(* CODESYS project XPlanarApplication.library
   Company: Beckhoff Automation LLC
   DefaultNamespace: XPlanarApplication
   Version: 1.0.1
   Placeholder: XPlanarApplication
   Title: XPlanarApplication

Project tree, tasks and I/O mapping:
  libraries: SPT Base Types, * (Beckhoff Automation LLC); SPT Event Logger, * (Beckhoff Automation LLC); Tc2_Math, * (Beckhoff Automation GmbH); Tc2_Standard, * (Beckhoff Automation GmbH); Tc2_System, * (Beckhoff Automation GmbH); Tc2_Utilities, * (Beckhoff Automation GmbH); Tc3_EventLogger, * (Beckhoff Automation GmbH); Tc3_Mc3PlanarMotion, * (Beckhoff Automation GmbH); Tc3_Physics, * (Beckhoff Automation GmbH); Tc3_XPlanarUtility, * (Beckhoff Automation GmbH)
  Mover/
    DUTs/
      data type ST_CommandLog
      data type ST_MoveDynamics
      data type ST_MoverCommand
      data type ST_MoverHMI
      data type ST_MoverObjectInfos
    TaskClasses/
      function block FB_AddToGroup [ST]: Execute
      function block FB_Disable [ST]: Execute
      function block FB_Enable [ST]: Execute
      function block FB_Halt [ST]: Execute
      function block FB_JoinClosestTrack [ST]: Execute, Update
      function block FB_JoinTrack [ST]: Execute
      function block FB_LeaveTrack [ST]: Execute
      function block FB_MoveA [ST]: Execute
      function block FB_MoveB [ST]: Execute
      function block FB_MoveToPosition [ST]: Execute
      function block FB_MoveZ [ST]: Execute
      function block FB_ResetMover [ST]: Execute
      function block FB_Rotate [ST]: Execute
      function block FB_SquareUp [ST]: Execute, Update
      function block FB_TrackMove [ST]: Execute
      function block FB_TrackMoveXY [ST]: Execute
    function block FB_XPlanarMover [ST]: FreeMove, JoinClosestTrack, JoinTrack, LeaveTrack, Rotate, SendToStation, SquareUp, TiltA, TiltB, TrackMove, TrackMoveXY, VerticalMove, Movement, Rotation, Tilt, ActualPosition, AddToGroup, CommandLog, Destination, Disable, Dynamics, Enable, Gap, Halt, IdentifiedBTN, InStation, MoveCommand, MoverBTN, MoverIndex, MoverType, pm, Reset, Status, Utility, CyclicLogic
    interface I_MoveCommands: FreeMove, JoinClosestTrack, JoinTrack, LeaveTrack, Rotate, SendToStation, SquareUp, TiltA, TiltB, TrackMove, TrackMoveXY, VerticalMove
    interface I_MoveDynamics: Movement, Rotation, Tilt
    interface I_XPlanarMover: ActualPosition, AddToGroup, CommandLog, Destination, Disable, Dynamics, Enable, Gap, Halt, IdentifiedBTN, InStation, MoveCommand, MoverBTN, MoverIndex, MoverType, pm, Reset, Status, Utility
  Part/
    Tasks/
      function block FB_AllowEnable [ST]: Execute
      function block FB_ForceDisable [ST]: Execute
      function block FB_Initialize [ST]: Execute
      function block FB_ResetPart [ST]: Execute
    function block FB_XPlanarPart [ST]: CyclicLogic, ForceDisable, Initialize, ObjectID, pm, Reset, SetAllowEnable, State
    interface I_XPlanarPart: ForceDisable, ObjectID, pm, Reset, SetAllowEnable, State
  Project Information/
    function F_GetCompany [ST]
    function F_GetTitle [ST]
    function F_GetVersion [ST]
  Station/
    DUT/
      data type E_StationType
      data type E_XplanarStationState
      data type ST_StationHMI
      data type ST_XPlanarStationObjectInfos
    function block FB_MoverQueue [ST]: Clear, Count, Dequeue, Enqueue, FirstMover, LastMover, MoverIDs, Queue
    function block FB_XPlanarStationBase [ST]: AllowQueing, CanReleaseMover, CurrentMover, Error, Execute, HasMover, ID, MoverDetected, MoverQueue, NextStation, NumMoversRequired, Position, Reset, Size, StationComplete, StationReady, StationType, TrackID, CyclicLogic, Name, WatchForMover
    interface I_XPlanarStation: AllowQueing, CanReleaseMover, CurrentMover, Execute, HasMover, ID, MoverQueue, Name, NextStation, NumMoversRequired, Position, Reset, Size, StationComplete, StationReady, StationType, TrackID
  Tile/
    DUT/
      data type ST_TileObjectInfos
      data type ST_TileTemperatures
    function block FB_XPlanarTile [ST]: Btn, CyclicLogic, DcLinkOk, Index, Initialize, PartIndex, PositionOnPart, Temperatures, TimeToShutdown, Update, Utility
    interface I_XPlanarTile: Btn, DcLinkOk, Index, PartIndex, PositionOnPart, Temperatures, TimeToShutdown, Update, Utility
  Track/
    DUT/
      data type E_TrackItemType
      data type ST_TrackDefinition
      data type ST_TrackItems
      data type ST_TrackStatus
    TaskClasses/
      function block FB_AddTrackToGroup [ST]: Execute
      function block FB_AppendLine [ST]: Execute
      function block FB_AppendPoint [ST]: Execute
      function block FB_BuildTrack [ST]: Execute, Update
      function block FB_ClearSegment [ST]: Execute
      function block FB_CloseLoop [ST]: Execute
      function block FB_DisableTrack [ST]: Execute
      function block FB_EnableTrack [ST]: Execute
      function block FB_SetEndAtTrack [ST]: Execute
      function block FB_SetStartFromTrack [ST]: Execute
      function block FB_TrackReset [ST]: Execute
    function block FB_XPlanarTrackSegment [ST]: AddToGroup, AppendLine, AppendPoint, Build, Clear, CloseLoop, Definition, Disable, Enable, GetTrackPositionAt, Index, MoverCount, MovingMoverCount, pm, Reset, SetEndAtTrack, SetStartFromTrack, Status, TrackLength, Utility, CyclicLogic
    interface I_XPlanarTrack: AddToGroup, AppendLine, AppendPoint, Build, Clear, CloseLoop, Definition, Disable, Enable, GetTrackPositionAt, Index, MoverCount, MovingMoverCount, pm, Reset, Status, TrackLength, Utility
  Version/
    global variables Global_Version
  XPlanarComponent/
    TaskClasses/
      function block FB_EnableGroup [ST]: Execute
      function block FB_MoverIdentification [ST]: Execute, Update
      function block FB_MoverRedetection [ST]: Execute, Update
      function block FB_ResetGroup [ST]: Execute
      function block FB_ResetXPlanar [ST]: Execute, Update
    function block FB_Component_XPlanar [ST]: CreateEvents, Monitoring, CyclicLogic, Abort, AddMoversToGroup, AddTracksToGroup, EnableGroup, EnableMovers, EnableTracks, IdentifyMovers, Initialize, MoverDetectionInfo, MoverRedetect, Reset, TileCount, TracksInitialized, Utility
  XPlanarResultClasses/
    function block FB_MoverTaskResult [ST]: Mover, Update, UpdateLog
    function block FB_PartTaskResult [ST]: Part
    function block FB_PlanarFeedbackResult [ST]: PlanarFeedback, Update
    function block FB_ResultBase [ST]: Aborted, BlockingObjectInfo, Busy, Done, Error, ErrorID, Result, TaskName
    function block FB_TrackTaskResult [ST]: Track
    interface I_PlanarTaskResult: Aborted, BlockingObjectInfo, Busy, Done, Error, ErrorID
  Class Diagram
  global variables ip
  00000000-0000-0000-0000-000000000000|LICENSE
  LICENSE
  global variables SystemParameters
  global variables XPlanar
  global variables XPlanarHMI
*)

// Mover/DUTs/ST_CommandLog
TYPE ST_CommandLog EXTENDS ST_MoverCommand :
	STRUCT
		Timestamp : STRING(24);
	END_STRUCT
END_TYPE

// Mover/DUTs/ST_MoveDynamics
TYPE ST_MoveDynamics :
STRUCT
	Velocity	: LREAL;
	Accel		: LREAL;
	Decel		: LREAL;
	Jerk		: LREAL;
END_STRUCT
END_TYPE

// Mover/DUTs/ST_MoverCommand
TYPE ST_MoverCommand :
	STRUCT
		Command : STRING;
		Vlocity : LREAL;
		Accel	: LREAL;
		Decel	: LREAL;
		Jerk	: LREAL;
	END_STRUCT
END_TYPE

// Mover/DUTs/ST_MoverHMI
TYPE ST_MoverHMI :
	STRUCT
		Enabled		   : BOOL;
		Error		   : BOOL;
		InStation	   : BOOL;
		ErrorID		   : UDINT;
		CurrentStation : STRING;
		CommandMode	   : STRING;
		LastCommand	   : STRING;
		EnableMover	   : BOOL;
		DisableMover   : BOOL;
		ResetMover	   : BOOL;
		HaltMover	   : BOOL;
	END_STRUCT
END_TYPE

// Mover/DUTs/ST_MoverObjectInfos
TYPE ST_MoverObjectInfos :
	STRUCT
		Width	 : DINT;
		Height	 : DINT;
		MoverBTN : STRING(13);
	END_STRUCT
END_TYPE

// Station/DUT/E_StationType
{attribute 'qualified_only'}
TYPE E_StationType : (
		Process		  := 0,
		DecisionPoint := 1,
		MultiMover	  := 2
	) UDINT;
END_TYPE

// Station/DUT/E_XplanarStationState
{attribute 'qualified_only'}
{attribute 'strict'}
{attribute 'to_string'}
TYPE E_XplanarStationState : (
		StationIdle := 0,
		ProcessMover,
		SquareUpMover,
		SendMoverAway,
		CycleComplete,
		SendQueue,
		StationError
	);
END_TYPE

// Station/DUT/ST_StationHMI
TYPE ST_StationHMI :
	STRUCT
		Error		   : BOOL;
		Reset		   : BOOL;
		StationReady   : BOOL;
		HasMover	   : BOOL;
		CurrentMoverID : STRING(13);
		CurrentState   : STRING;
	END_STRUCT
END_TYPE

// Station/DUT/ST_XPlanarStationObjectInfos
TYPE ST_XPlanarStationObjectInfos :
	STRUCT
		X	   : DINT;
		Y	   : DINT;
		Width  : DINT;
		Height : DINT;
	END_STRUCT
END_TYPE

// Tile/DUT/ST_TileObjectInfos
TYPE ST_TileObjectInfos :
	STRUCT
		X	   : DINT;
		Y	   : DINT;
		Width  : DINT;
		Height : DINT;
	END_STRUCT
END_TYPE

// Tile/DUT/ST_TileTemperatures
TYPE ST_TileTemperatures :
	STRUCT
		Center : LREAL;
		East   : LREAL;
		West   : LREAL;
		North  : LREAL;
		South  : LREAL;
	END_STRUCT
END_TYPE

// Track/DUT/E_TrackItemType
TYPE E_TrackItemType :
(
	Point := 0,
	Line,
	Circle
);
END_TYPE

// Track/DUT/ST_TrackDefinition
TYPE ST_TrackDefinition :
	STRUCT
		StartFromTrackID : UDINT;
		EndAtTrackID	 : UDINT;
		CloseLoop		 : BOOL;
		Items			 : ARRAY[1..SystemParameters.MAX_OBJECTS_PER_TRACK] OF ST_TrackItems;
	END_STRUCT
END_TYPE

// Track/DUT/ST_TrackItems
TYPE ST_TrackItems :
STRUCT
	ItemType		: E_TrackItemType;
	StartPoint		: PositionXYC;
	EndPoint		: PositionXYC;
	CenterPoint		: PositionXY;
	CircleClockwise : BOOL;
END_STRUCT
END_TYPE

// Track/DUT/ST_TrackStatus
TYPE ST_TrackStatus :
	STRUCT
		State			 : MC_PLANAR_STATE;
		OperationMode	 : MC_PLANAR_TRACK_OPERATION_MODE;
		MoverCount		 : UDINT;
		CalculatedLength : LREAL;
	END_STRUCT
END_TYPE

// Version/Global_Version
{attribute 'TcGenerated'}
{attribute 'no-analysis'}
{attribute 'linkalways'}
// This function has been automatically generated from the project information.
VAR_GLOBAL CONSTANT
	{attribute 'const_non_replaced'}
	stLibVersion_XPlanarApplication : ST_LibVersion := (iMajor := 1, iMinor := 0, iBuild := 1, iRevision := 0, nFlags := 1, sVersion := '1.0.1');
END_VAR

// ip
{attribute 'qualified_only'}
VAR_GLOBAL
	Movers	 : ARRAY[0..SystemParameters.MOVER_COUNT] OF I_XPlanarMover;
	Tracks	 : ARRAY[0..SystemParameters.TRACK_COUNT] OF I_XPlanarTrack;
	Stations : ARRAY[0..SystemParameters.STATION_COUNT] OF I_XPlanarStation;
END_VAR

// SystemParameters
{attribute 'qualified_only'}
VAR_GLOBAL CONSTANT
	EnableCommandTracing  : BOOL  := FALSE; //Enables mover command trace logging
	AssumedMoverSize	  : LREAL := 50;
	MAX_LOG_COUNT		  : UINT  := 20; //Size of command mover log
	MOVER_COUNT			  : UINT  := 4;	 //Total number of movers configured in the system
	TRACK_COUNT			  : UINT  := 1;	 //Total number of track segments in the system
	MAX_OBJECTS_PER_TRACK : UINT  := 20; //Maximum number of points or lines defined in a single track segment
	STATION_COUNT		  : UINT  := 3;	 //Total number of stations in the system
	MaxMoversPerStation	  : UDINT := 4;	 //Max number of movers allowed to queue in a station 
	TileDiagUpdate		  : LREAL := 0;	 //Tile Diagnostic data update rate in seconds.  Set to 0 to disable
END_VAR

// XPlanar
{attribute 'qualified_only'}
VAR_GLOBAL
	Environment		: Tc3_MC3PlanarMotion.MC_PlanarEnvironment;
	Group			: Tc3_MC3PlanarMotion.MC_PlanarGroup;
	EnvironmentTcIo : Tc3_XPlanarUtility.FB_TcIoXPlanarEnvironment;
	OperationMode	: XPlanarOperationMode;
	XPUCount		: UINT;
	PartCount		: UINT;
	TrackCount		: UINT;
	MoverCount		: UINT;
	TileCount		: UINT;

END_VAR

// XPlanarHMI
{attribute 'qualified_only'}
VAR_GLOBAL
	MoverObjects	: ARRAY[1..SystemParameters.MOVER_COUNT] OF ST_MoverObjectInfos;
	MoverPositions	: ARRAY[1..SystemParameters.MOVER_COUNT] OF MoverVector;
	TileObjects		: ARRAY[1..Param_TcIoXPlanarEnvironment.MaxTiles] OF ST_TileObjectInfos;
	StationObjects	: ARRAY[1..SystemParameters.STATION_COUNT] OF ST_XPlanarStationObjectInfos;
END_VAR

// Mover/TaskClasses/FB_AddToGroup
FUNCTION_BLOCK FB_AddToGroup EXTENDS FB_MoverTaskResult
VAR
END_VAR

METHOD Execute : I_PlanarTaskResult
VAR_INPUT
	Group : REFERENCE TO MC_PlanarGroup;
END_VAR
IF NOT HasRun THEN
	_Done	 := FALSE;
	_Error	 := FALSE;
	_Busy	 := FALSE;
	_ErrorID := 0;
	ipMover.pm.AddToGroup(_PlanarFb, Group);

	//Update mover command log				
	LogEntry.Command := CONCAT('AddMoverToGroup ', TO_STRING(Group.MCTOPLC_STD.GroupOID));
	LogEntry.Accel	 := 0;
	LogEntry.Decel	 := 0;
	LogEntry.Jerk	 := 0;
	LogEntry.Vlocity := 0;
	UpdateLog();
	HasRun := TRUE;
END_IF

Execute := THIS^;

//Heartbeat that the method is active
ExecuteWatchdog := ExecuteWatchdog + 1;
END_METHOD

END_FUNCTION_BLOCK

// XPlanarResultClasses/FB_MoverTaskResult
FUNCTION_BLOCK FB_MoverTaskResult EXTENDS FB_PlanarFeedbackResult
VAR
	ipMover : I_XPlanarMover;

	//CmdLog		   : REFERENCE TO ARRAY[0..SystemParameters.MAX_LOG_COUNT] OF ST_CommandLog;
	GetTime		   : GETSYSTEMTIME;
	SysTime		   : T_FILETIME;
	LogEntry	   : ST_MoverCommand;
	ActualPosition : MoverVector;
	RT_ADSWarn	   : R_Trig;
	MoverStr	   : STRING;
END_VAR

PROPERTY Mover : I_XPlanarMover
SET
ipMover := Mover;
END_SET
END_PROPERTY

METHOD Update
ActualPosition := ipMover.ActualPosition;
SUPER^.Update();
RT_ADSWarn(CLK := _PlanarFb.Error);
IF RT_ADSWarn.Q THEN
	MoverStr := CONCAT('Mover ', TO_STRING(ipMover.MoverIndex));
	ADSLOGSTR(ADSLOG_MSGTYPE_WARN, CONCAT(MoverStr, ' : %s'), CONCAT(_TaskName, CONCAT('Error ', TO_STRING(_PlanarFb.ErrorId))));
END_IF
END_METHOD

METHOD UpdateLog
VAR_INST
	i : UINT;
END_VAR
IF SystemParameters.MAX_LOG_COUNT > 0 THEN
	FOR i := SystemParameters.MAX_LOG_COUNT - 1 TO 1 BY -1 DO
		IF i < SystemParameters.MAX_LOG_COUNT THEN
			ipMover.CommandLog[i + 1] := ipMover.CommandLog[i];
		END_IF
	END_FOR

	ipMover.CommandLog[1] := ipMover.CommandLog[0];
	GetTime(timeLoDW => SysTime.dwLowDateTime, timeHiDW => SysTime.dwHighDateTime);
	ipMover.CommandLog[0].Timestamp := SYSTEMTIME_TO_STRING(FILETIME_TO_SYSTEMTIME(SysTime));
	ipMover.CommandLog[0].Command	:= LogEntry.Command;
	ipMover.CommandLog[0].Accel		:= LogEntry.Accel;
	ipMover.CommandLog[0].Decel		:= LogEntry.Decel;
	ipMover.CommandLog[0].Jerk		:= LogEntry.Jerk;
	ipMover.CommandLog[0].Vlocity	:= LogEntry.Vlocity;
END_IF
END_METHOD

END_FUNCTION_BLOCK

// XPlanarResultClasses/FB_PlanarFeedbackResult
FUNCTION_BLOCK FB_PlanarFeedbackResult EXTENDS FB_ResultBase
VAR
	_PlanarFb		: MC_PlanarFeedback;
	HasRun			: BOOL;
	ExecuteWatchdog : UDINT;
	TaskState		: UDINT;
END_VAR

PROPERTY PlanarFeedback : REFERENCE TO MC_PlanarFeedback
GET
PlanarFeedback ref= _PlanarFb;
END_GET
END_PROPERTY

METHOD Update
VAR_INST
	WatchdogCheck : UDINT;
END_VAR
//Update Command Feedback Status
_PlanarFb.Update();

//Update Interface based on Command Feedback status
_Aborted			:= _PlanarFb.Aborted;
_Busy				:= _PlanarFb.Active OR _PlanarFb.Busy;
_Done				:= _PlanarFb.Done;
_Error				:= _PlanarFb.Error;
_ErrorID			:= _PlanarFb.ErrorId;
_BlockingObjectInfo := _PlanarFb.objectInfo;

//Heartbeat to know execute is active
IF ExecuteWatchdog <> WatchdogCheck THEN
	WatchdogCheck := ExecuteWatchdog;
ELSE
	HasRun			:= FALSE;
	ExecuteWatchdog := 0;
END_IF
END_METHOD

END_FUNCTION_BLOCK

// XPlanarResultClasses/FB_ResultBase
FUNCTION_BLOCK FB_ResultBase EXTENDS FB_BaseFB IMPLEMENTS I_PlanarTaskResult
VAR
	_TaskName			: STRING;
	_Done				: BOOL;
	_Aborted			: BOOL;
	_BlockingObjectInfo : PlanarObjectInfo;
END_VAR

PROPERTY Aborted : BOOL
GET
Aborted := _Aborted;
END_GET
SET
_Aborted := Aborted;
END_SET
END_PROPERTY

PROPERTY BlockingObjectInfo : REFERENCE TO Tc3_Mc3PlanarMotion.PlanarObjectInfo
GET
BlockingObjectInfo ref= _BlockingObjectInfo;
END_GET
END_PROPERTY

PROPERTY Busy : BOOL
GET
Busy := _Busy;
END_GET
SET
_Busy := Busy;
END_SET
END_PROPERTY

PROPERTY Done : BOOL
GET
Done := _Done;
END_GET
SET
_Done := Done;
END_SET
END_PROPERTY

PROPERTY Error : BOOL
GET
Error := _Error;
END_GET
SET
_Error := Error;
END_SET
END_PROPERTY

PROPERTY ErrorID : UDINT
GET
ErrorID := _ErrorID;
END_GET
SET
_ErrorID := ErrorID;
END_SET
END_PROPERTY

PROPERTY Result : I_PlanarTaskResult
GET
Result := THIS^;
END_GET
END_PROPERTY

PROPERTY TaskName : STRING
GET
TaskName := _TaskName;
END_GET
SET
_TaskName := TaskName;
END_SET
END_PROPERTY

END_FUNCTION_BLOCK

// XPlanarResultClasses/I_PlanarTaskResult
INTERFACE I_PlanarTaskResult

PROPERTY Aborted : BOOL
GET
END_GET
END_PROPERTY

PROPERTY BlockingObjectInfo : REFERENCE TO PlanarObjectInfo
GET
END_GET
END_PROPERTY

PROPERTY Busy : BOOL
GET
END_GET
END_PROPERTY

PROPERTY Done : BOOL
GET
END_GET
END_PROPERTY

PROPERTY Error : BOOL
GET
END_GET
END_PROPERTY

PROPERTY ErrorID : UDINT
GET
END_GET
END_PROPERTY

END_INTERFACE

// Mover/I_XPlanarMover
INTERFACE I_XPlanarMover EXTENDS I_BaseFb

PROPERTY ActualPosition : REFERENCE TO MoverVector
GET
END_GET
END_PROPERTY

METHOD AddToGroup : I_PlanarTaskResult
VAR_INPUT
	PlanarGroup : REFERENCE TO MC_PlanarGroup;
END_VAR
END_METHOD

PROPERTY CommandLog : REFERENCE TO ARRAY [0..SystemParameters.MAX_LOG_COUNT] of ST_CommandLog
GET
END_GET
END_PROPERTY

PROPERTY Destination : I_XPlanarStation
GET
END_GET
SET
END_SET
END_PROPERTY

METHOD Disable : I_PlanarTaskResult
END_METHOD

PROPERTY Dynamics : I_MoveDynamics
GET
END_GET
END_PROPERTY

METHOD Enable : I_PlanarTaskResult
END_METHOD

PROPERTY Gap : LREAL
GET
END_GET
SET
END_SET
END_PROPERTY

METHOD Halt : I_PlanarTaskResult
END_METHOD

PROPERTY IdentifiedBTN : STRING
GET
END_GET
END_PROPERTY

PROPERTY InStation : BOOL
GET
END_GET
SET
END_SET
END_PROPERTY

PROPERTY MoveCommand : I_MoveCommands
GET
END_GET
END_PROPERTY

PROPERTY MoverBTN : STRING
GET
END_GET
END_PROPERTY

PROPERTY MoverIndex : UDINT
GET
END_GET
SET
END_SET
END_PROPERTY

PROPERTY MoverType : XplanarMoverType
GET
END_GET
SET
END_SET
END_PROPERTY

PROPERTY pm : REFERENCE TO MC_PlanarMover
GET
END_GET
END_PROPERTY

//! @summary Clears error flags and error IDs for this component
{attribute 'TcRpcEnable'}
METHOD PUBLIC Reset : I_PlanarTaskResult
END_METHOD

PROPERTY Status : REFERENCE TO CDT_MCTOPLC_PLANAR_MOVER_STD
GET
END_GET
END_PROPERTY

PROPERTY Utility : I_TcIoXPlanarMover
GET
END_GET
SET
END_SET
END_PROPERTY

END_INTERFACE

// Station/I_XPlanarStation
INTERFACE I_XPlanarStation EXTENDS I_BaseFb

PROPERTY AllowQueing : BOOL
GET
END_GET
SET
END_SET
END_PROPERTY

PROPERTY CanReleaseMover : BOOL
SET
END_SET
END_PROPERTY

PROPERTY CurrentMover : I_XPlanarMover
GET
END_GET
END_PROPERTY

METHOD Execute
END_METHOD

PROPERTY HasMover : BOOL
GET
END_GET
SET
END_SET
END_PROPERTY

PROPERTY ID : UDINT
GET
END_GET
SET
END_SET
END_PROPERTY

PROPERTY MoverQueue : REFERENCE TO FB_MoverQueue
GET
END_GET
END_PROPERTY

PROPERTY Name : STRING
GET
END_GET
SET
END_SET
END_PROPERTY

PROPERTY NextStation : I_XPlanarStation
GET
END_GET
SET
END_SET
END_PROPERTY

PROPERTY NumMoversRequired : UDINT
GET
END_GET
SET
END_SET
END_PROPERTY

PROPERTY Position : REFERENCE TO PositionXYC
GET
END_GET
END_PROPERTY

METHOD Reset : BOOL
END_METHOD

PROPERTY Size : REFERENCE TO Position2D_LREAL
GET
END_GET
END_PROPERTY

PROPERTY StationComplete : BOOL
SET
END_SET
END_PROPERTY

PROPERTY StationReady : BOOL
GET
END_GET
END_PROPERTY

PROPERTY StationType : E_StationType
GET
END_GET
SET
END_SET
END_PROPERTY

PROPERTY TrackID : UDINT
GET
END_GET
SET
END_SET
END_PROPERTY

END_INTERFACE

// Station/FB_MoverQueue
//=============================================================================

//	FB_MoverQueue

//=============================================================================

//

//	FIFO Queue for use by stations

//

//-----------------------------------------------------------------------------
FUNCTION_BLOCK FB_MoverQueue
VAR
	MoversInQueue : UDINT := 0;
	ipMovers	  : ARRAY[1..SystemParameters.MaxMoversPerStation] OF I_XPlanarMover;
END_VAR

//=============================================================================

//	Method Clear()

//=============================================================================

//

//	Brute force reset of buffer

//

//-----------------------------------------------------------------------------
METHOD Clear : BOOL
MEMSET(ADR(ipMovers), 0, SIZEOF(ipMovers));
MoversInQueue := 0;
Clear		  := TRUE;
END_METHOD

PROPERTY Count : UDINT
GET
VAR
	i	 : UDINT;
	temp : UDINT;
END_VAR
Count := MoversInQueue;
END_GET
END_PROPERTY

METHOD Dequeue : BOOL
IF MoversInQueue > 0 THEN
	ipMovers[1].InStation := FALSE;
	MEMSET(ADR(ipMovers[1]), 0, SIZEOF(ipMovers[1]));
	MoversInQueue := MoversInQueue - 1;
	IF MoversInQueue > 0 THEN
		MEMMOVE(ADR(ipMovers[1]), ADR(ipMovers[2]), SIZEOF(ipMovers[2]) * MoversInQueue);
		MEMSET(ADR(ipMovers[MoversInQueue + 1]), 0, (SIZEOF(ipMovers[1]) * (SystemParameters.MaxMoversPerStation - MoversInQueue)));
	END_IF

	Dequeue := TRUE;
END_IF
END_METHOD

METHOD Enqueue : BOOL
VAR_INPUT
	ipMover : I_XPlanarMover;
END_VAR
IF MoversInQueue < SystemParameters.MaxMoversPerStation THEN
	MoversInQueue			:= MoversInQueue + 1;
	ipMover.InStation		:= TRUE;
	ipMovers[MoversInQueue] := ipMover;
	Enqueue					:= TRUE;
END_IF
END_METHOD

PROPERTY FirstMover : I_XPlanarMover
GET
IF MoversInQueue > 0 THEN
	FirstMover := ipMovers[1];
END_IF
END_GET
END_PROPERTY

PROPERTY LastMover : I_XPlanarMover
GET
IF MoversInQueue > 0 THEN
	LastMover := ipMovers[MoversInQueue];
END_IF
END_GET
END_PROPERTY

PROPERTY MoverIDs : ARRAY[1..SystemParameters.MaxMoversPerStation] OF UDINT
GET
VAR
	i : UDINT;
END_VAR
FOR i := 1 TO MoversInQueue DO
	IF ipMovers[i] <> 0 THEN
		MoverIDs[i] := ipMovers[i].MoverIndex;
	END_IF
END_FOR
END_GET
END_PROPERTY

PROPERTY Queue : REFERENCE TO ARRAY[1..SystemParameters.MaxMoversPerStation] OF I_XPlanarMover;
GET
VAR
	i : UDINT;
END_VAR
Queue ref= ipMovers;
END_GET
END_PROPERTY

END_FUNCTION_BLOCK

// Mover/I_MoveDynamics
INTERFACE I_MoveDynamics EXTENDS __SYSTEM.IQueryInterface

PROPERTY Movement : REFERENCE TO ST_MoveDynamics
GET
END_GET
END_PROPERTY

PROPERTY Rotation : REFERENCE TO ST_MoveDynamics
GET
END_GET
END_PROPERTY

PROPERTY Tilt : REFERENCE TO ST_MoveDynamics
GET
END_GET
END_PROPERTY

END_INTERFACE

// Mover/I_MoveCommands
INTERFACE I_MoveCommands EXTENDS __SYSTEM.IQueryInterface

METHOD FreeMove : I_PlanarTaskResult
VAR_INPUT
	XPosition : LREAL;
	YPosition : LREAL;
END_VAR
END_METHOD

{attribute 'TcRpcEnable'}
METHOD JoinClosestTrack : I_PlanarTaskResult
VAR_INPUT
	UseOrientation : BOOL;
END_VAR
END_METHOD

{attribute 'TcRpcEnable'}
METHOD JoinTrack : I_PlanarTaskResult
VAR_INPUT
	ipTrack		   : I_XPlanarTrack;
	UseOrientation : BOOL;
END_VAR
END_METHOD

{attribute 'TcRpcEnable'}
METHOD LeaveTrack : I_PlanarTaskResult
VAR_INPUT
	DestinationX   : LREAL;
	DestinationY   : LREAL;
	UseOrientation : BOOL;
END_VAR
END_METHOD

{attribute 'TcRpcEnable'}
METHOD Rotate : I_PlanarTaskResult
VAR_INPUT
	Position		: LREAL;
	AdditionalTurns : DINT;
END_VAR
END_METHOD

{attribute 'TcRpcEnable'}
METHOD SendToStation : I_PlanarTaskResult
VAR_INPUT
	Destination : I_XPlanarStation;
END_VAR
END_METHOD

{attribute 'TcRpcEnable'}
METHOD SquareUp : I_PlanarTaskResult
END_METHOD

METHOD TiltA : I_PlanarTaskResult
VAR_INPUT
	Position : LREAL;
END_VAR
END_METHOD

METHOD TiltB : I_PlanarTaskResult
VAR_INPUT
	Position : LREAL;
END_VAR
END_METHOD

{attribute 'TcRpcEnable'}
METHOD TrackMove : I_PlanarTaskResult
VAR_INPUT
	Position : LREAL;
	Gap		  : LREAL;
	Track	  : I_XPlanarTrack;
	Direction : Tc3_Mc3PlanarMotion.MC_DIRECTION;
END_VAR
END_METHOD

{attribute 'TcRpcEnable'}
METHOD TrackMoveXY : I_PlanarTaskResult
VAR_INPUT
	XPosition : LREAL;
	YPosition : LREAL;
	Gap		  : LREAL;
	Track	  : I_XPlanarTrack;
	Direction : Tc3_Mc3PlanarMotion.MC_DIRECTION;
END_VAR
END_METHOD

{attribute 'TcRpcEnable'}
METHOD VerticalMove : I_PlanarTaskResult
VAR_INPUT
	Position : LREAL;
END_VAR
END_METHOD

END_INTERFACE

// Track/I_XPlanarTrack
INTERFACE I_XPlanarTrack EXTENDS I_BaseFb

METHOD AddToGroup : I_PlanarTaskResult
VAR_INPUT
	PlanarGroup : REFERENCE TO MC_PlanarGroup;
END_VAR
END_METHOD

METHOD AppendLine : I_PlanarTaskResult
VAR_INPUT
	StartPointX : LREAL;
	StartPointY : LREAL;
	EndPointX	: LREAL;
	EndPointY	: LREAL;
END_VAR
END_METHOD

METHOD AppendPoint : I_PlanarTaskResult
VAR_INPUT
	XPoint : LREAL;
	YPoint : LREAL;
END_VAR
END_METHOD

METHOD Build : I_PlanarTaskResult
END_METHOD

METHOD Clear : I_PlanarTaskResult
END_METHOD

METHOD CloseLoop : I_PlanarTaskResult
END_METHOD

PROPERTY Definition : REFERENCE TO ST_TrackDefinition
GET
END_GET
END_PROPERTY

METHOD Disable : I_PlanarTaskResult
END_METHOD

{attribute 'TcRpcEnable'}
METHOD Enable : I_PlanarTaskResult
END_METHOD

METHOD GetTrackPositionAt : LREAL;
VAR_IN_OUT
	Position : PositionXYC;
END_VAR
END_METHOD

PROPERTY Index : UDINT
GET
END_GET
SET
END_SET
END_PROPERTY

PROPERTY MoverCount : UDINT
GET
END_GET
END_PROPERTY

PROPERTY MovingMoverCount : UDINT
GET
END_GET
END_PROPERTY

PROPERTY pm : REFERENCE TO MC_PlanarTrack
GET
END_GET
END_PROPERTY

METHOD Reset : I_PlanarTaskResult
VAR_INPUT
END_VAR
END_METHOD

PROPERTY Status : REFERENCE TO CDT_MCTOPLC_PLANAR_TRACK
GET
END_GET
END_PROPERTY

PROPERTY TrackLength : LREAL
GET
END_GET
END_PROPERTY

PROPERTY Utility : I_McPlanarTrack
GET
END_GET
END_PROPERTY

END_INTERFACE

// Mover/TaskClasses/FB_Disable
FUNCTION_BLOCK FB_Disable EXTENDS FB_MoverTaskResult
VAR
END_VAR

METHOD Execute : I_PlanarTaskResult
VAR_INPUT
END_VAR
IF NOT HasRun AND ipMover.Status.State <> MC_Planar_State.Disabled THEN
	_Done	 := FALSE;
	_Error	 := FALSE;
	_Busy	 := FALSE;
	_ErrorID := 0;
	ipMover.pm.Disable(_PlanarFb);

	//Update mover command log				
	LogEntry.Command := 'DisableMover';
	LogEntry.Accel	 := 0;
	LogEntry.Decel	 := 0;
	LogEntry.Jerk	 := 0;
	LogEntry.Vlocity := 0;
	UpdateLog();
	HasRun := TRUE;
END_IF

Execute := THIS^;

//Heartbeat that the method is active
ExecuteWatchdog := ExecuteWatchdog + 1;
END_METHOD

END_FUNCTION_BLOCK

// Mover/TaskClasses/FB_Enable
FUNCTION_BLOCK FB_Enable EXTENDS FB_MoverTaskResult
VAR
END_VAR

METHOD Execute : I_PlanarTaskResult
IF NOT HasRun AND ipMover.Status.State = MC_Planar_State.Disabled THEN
	_Done	 := FALSE;
	_Error	 := FALSE;
	_Busy	 := FALSE;
	_ErrorID := 0;
	ipMover.pm.Enable(_PlanarFb);

	//Update mover command log				
	LogEntry.Command := 'EnableMover';
	LogEntry.Accel	 := 0;
	LogEntry.Decel	 := 0;
	LogEntry.Jerk	 := 0;
	LogEntry.Vlocity := 0;
	UpdateLog();
	HasRun := TRUE;
END_IF

Execute := THIS^;

//Heartbeat that the method is active
ExecuteWatchdog := ExecuteWatchdog + 1;
END_METHOD

END_FUNCTION_BLOCK

// Mover/TaskClasses/FB_Halt
FUNCTION_BLOCK FB_Halt EXTENDS FB_MoverTaskResult
VAR
	BusyStatus : MoverBusy;
END_VAR

METHOD Execute : I_PlanarTaskResult
VAR_INPUT
	Dynamics : DynamicConstraint_PathXYZ;
END_VAR
BusyStatus := ipMover.Status.Busy;
IF NOT HasRun AND BusyStatus.busyMover THEN
	_Done	 := FALSE;
	_Error	 := FALSE;
	_Busy	 := FALSE;
	_ErrorID := 0;
	ipMover.pm.Halt(_PlanarFb, Dynamics);

	//Update mover command log				
	LogEntry.Command := 'HaltMover';
	LogEntry.Accel	 := Dynamics.A;
	LogEntry.Decel	 := Dynamics.D;
	LogEntry.Jerk	 := Dynamics.J;
	LogEntry.Vlocity := Dynamics.V;
	UpdateLog();
	HasRun := TRUE;
END_IF

Execute := THIS^;

//Heartbeat that the method is active
ExecuteWatchdog := ExecuteWatchdog + 1;
END_METHOD

END_FUNCTION_BLOCK

// Mover/TaskClasses/FB_JoinClosestTrack
FUNCTION_BLOCK FB_JoinClosestTrack EXTENDS FB_MoverTaskResult
VAR
	JoinTrackOptions	 : ST_JoinTrackOptions;
	TrackJoinDistances	 : ARRAY[1..SystemParameters.TRACK_COUNT] OF LREAL;
	_UseOrientation		 : BOOL;
	_MoveDynamics		 : DynamicConstraint_PathXYZ;
	i					 : UINT;
	MoverSetPosition	 : MoverVector;
	MoverCurrentPosition : PositionXYC;
	MoverJoinPosition	 :  ARRAY[1..SystemParameters.TRACK_COUNT] OF PositionXYC;
	MoverArcPosition	 :  ARRAY[1..SystemParameters.TRACK_COUNT] OF LREAL;
	ShortestDistance	 : LREAL;
	TrackToJoin			 : UINT;
	Join				 : BOOL;
END_VAR

METHOD Execute : I_PlanarTaskResult
VAR_INPUT
	UseOrientation : BOOL;
	MoveDynamics   : DynamicConstraint_PathXYZ;
END_VAR
IF NOT HasRun AND (ipMover.Status.CommandMode <> MC_Planar_Mover_Command_Mode.OnTrack) THEN
	_Done			:= FALSE;
	_Error			:= FALSE;
	_Busy			:= FALSE;
	_ErrorID		:= 0;
	_UseOrientation := UseOrientation;
	_MoveDynamics	:= MoveDynamics;
	Join			:= TRUE;
	HasRun			:= TRUE;
END_IF

Execute := THIS^;

//Heartbeat that the method is active
ExecuteWatchdog := ExecuteWatchdog + 1;
END_METHOD

METHOD Update
VAR_INST
	WatchdogCheck : UDINT;
END_VAR
//***Overwriting the update method because this task contains a state machine that must be monitored cyclically.***
_PlanarFb.Update();

//State logic for the task
CASE TaskState OF
	0: // Init
		_Busy := FALSE;
		IF Join THEN
			_Done			 := FALSE;
			_Error			 := FALSE;
			_ErrorID		 := 0;
			_Busy			 := TRUE;
			Join			 := FALSE;
			ShortestDistance := 0;
			TaskState		 := TaskState + 10;
		END_IF

	10: //Resolve Mover Position
		MoverSetPosition	   := ipMover.pm.MCTOPLC.SET.SetPos;
		MoverCurrentPosition.x := MoverSetPosition.x;
		MoverCurrentPosition.y := MoverSetPosition.y;
		MoverCurrentPosition.c := MoverSetPosition.c;
		TaskState			   := TaskState + 10;

	20: //Calculate distance from tracks
		FOR i := 1 TO SystemParameters.TRACK_COUNT DO
			//Get arc position based on mover position
			MoverArcPosition[i] := ip.Tracks[i].GetTrackPositionAt(MoverCurrentPosition);

			//Get Position based on arc position
			ip.Tracks[i].pm.GetPositionAt(MoverArcPosition[i], MoverJoinPosition[i]);

			//Save position delta
			TrackJoinDistances[i] := ABS(MoverJoinPosition[i].x - MoverCurrentPosition.x) + ABS(MoverJoinPosition[i].y - MoverCurrentPosition.y);
		END_FOR

		TaskState := TaskState + 10;

	30: //Find Closest Track
		FOR i := 1 TO SystemParameters.TRACK_COUNT DO
			IF ShortestDistance = 0 OR TrackJoinDistances[i] < ShortestDistance THEN
				ShortestDistance := TrackJoinDistances[i];
				TrackToJoin		 := i;
			END_IF
		END_FOR

		TaskState := TaskState + 10;

	40: //Join the closest track
		JoinTrackOptions.useOrientation := _UseOrientation;
		ipMover.pm.JoinTrack(_PlanarFb,
							 ip.Tracks[TrackToJoin].pm,
							 _MoveDynamics,
							 JoinTrackOptions);

		//Update mover command log				
		LogEntry.Command := CONCAT('JoinClosestTrack : ', TO_STRING(TrackToJoin));
		LogEntry.Accel	 := _MoveDynamics.A;
		LogEntry.Decel	 := _MoveDynamics.D;
		LogEntry.Jerk	 := _MoveDynamics.J;
		LogEntry.Vlocity := _MoveDynamics.V;
		UpdateLog();
		TaskState := TaskState + 10;

	50: //Watch feedback
		IF _PlanarFb.Done THEN
			TaskState := 60;
		ELSIF _PlanarFb.Error THEN
			_Error				:= TRUE;
			_ErrorID			:= _PlanarFb.ErrorId;
			_BlockingObjectInfo := _PlanarFb.objectInfo;
			TaskState			:= 0;
		END_IF

	60: //Task Complete
		THIS^._Done := TRUE;
		TaskState	:= 0;
END_CASE

RT_ADSWarn(CLK := _PlanarFb.Error);
IF RT_ADSWarn.Q THEN
	ADSLOGSTR(ADSLOG_MSGTYPE_WARN, CONCAT('Mover ', ipMover.MoverBTN), CONCAT(_TaskName, CONCAT('Error ', TO_STRING(_PlanarFb.ErrorId))));
END_IF

IF ExecuteWatchdog <> WatchdogCheck THEN
	WatchdogCheck := ExecuteWatchdog;
ELSE
	HasRun			:= FALSE;
	ExecuteWatchdog := 0;
END_IF
END_METHOD

END_FUNCTION_BLOCK

// Mover/TaskClasses/FB_JoinTrack
FUNCTION_BLOCK FB_JoinTrack EXTENDS FB_MoverTaskResult
VAR
	JoinTrackOptions : ST_JoinTrackOptions;
END_VAR

METHOD Execute : I_PlanarTaskResult
VAR_INPUT
	ipTrack		   : I_XPlanarTrack;
	UseOrientation : BOOL;
	MoveDynamics   : DynamicConstraint_PathXYZ;
END_VAR
IF NOT HasRun AND (ipMover.Status.CommandMode <> MC_Planar_Mover_Command_Mode.OnTrack) THEN
	_Done	 := FALSE;
	_Error	 := FALSE;
	_Busy	 := FALSE;
	_ErrorID := 0;
	JoinTrackOptions.useOrientation := UseOrientation;
	ipMover.pm.JoinTrack(_PlanarFb,
					ipTrack.pm,
					MoveDynamics,
					JoinTrackOptions);

	//Update mover command log				
	LogEntry.Command := CONCAT('JoinTrack : ', TO_STRING(ipTrack.Index));
	LogEntry.Accel	 := MoveDynamics.A;
	LogEntry.Decel	 := MoveDynamics.D;
	LogEntry.Jerk	 := MoveDynamics.J;
	LogEntry.Vlocity := MoveDynamics.V;
	UpdateLog();
	HasRun := TRUE;
END_IF

Execute := THIS^;

//Heartbeat that the method is active
ExecuteWatchdog := ExecuteWatchdog + 1;
END_METHOD

END_FUNCTION_BLOCK

// Mover/TaskClasses/FB_LeaveTrack
FUNCTION_BLOCK FB_LeaveTrack EXTENDS FB_MoverTaskResult
VAR
	LeaveTrackOptions : ST_LeaveTrackOptions;
END_VAR

METHOD Execute : I_PlanarTaskResult
VAR_INPUT
	TargetPositionX : LREAL;
	TargetPositionY : LREAL;
	UseOrientation	: BOOL;
	MoveDynamics	: DynamicConstraint_PathXYZ;
END_VAR

VAR_INST
	Target : PositionXYC;
END_VAR
IF NOT HasRun AND ipMover.Status.CommandMode = MC_Planar_Mover_Command_Mode.OnTrack THEN
	_Done							 := FALSE;
	_Error							 := FALSE;
	_Busy							 := FALSE;
	_ErrorID						 := 0;
	LeaveTrackOptions.useOrientation := UseOrientation;
	Target.SetValuesXYC(TargetPositionX, TargetPositionY, ActualPosition.c);
	ipMover.pm.LeaveTrack(_PlanarFb,
						  Target,
						  MoveDynamics,
						  LeaveTrackOptions);

	//Update mover command log				
	LogEntry.Command := CONCAT('LeaveTrackTo : ', CONCAT(CONCAT('X= ', TO_STRING(TargetPositionX)), CONCAT(' Y= ', TO_STRING(TargetPositionY))));
	LogEntry.Accel	 := MoveDynamics.A;
	LogEntry.Decel	 := MoveDynamics.D;
	LogEntry.Jerk	 := MoveDynamics.J;
	LogEntry.Vlocity := MoveDynamics.V;
	UpdateLog();
	HasRun := TRUE;
END_IF

Execute := THIS^;

//Heartbeat that the method is active
ExecuteWatchdog := ExecuteWatchdog + 1;
END_METHOD

END_FUNCTION_BLOCK

// Mover/TaskClasses/FB_MoveA
FUNCTION_BLOCK FB_MoveA EXTENDS FB_MoverTaskResult
VAR
END_VAR

METHOD Execute : I_PlanarTaskResult
VAR_INPUT
	Position	 : LREAL;
	MoveDynamics : DynamicConstraint_Coordinates;
END_VAR
IF NOT HasRun THEN
	_Done	 := FALSE;
	_Error	 := FALSE;
	_Busy	 := FALSE;
	_ErrorID := 0;
	ipMover.pm.MoveA(_PlanarFb, Position, MoveDynamics);

	//Update mover command log				
	LogEntry.Command := CONCAT('MoveA : ', TO_STRING(Position));
	LogEntry.Accel	 := MoveDynamics.GetA(Coord_Mcs_A1);
	LogEntry.Decel	 := MoveDynamics.GetD(Coord_Mcs_A1);
	LogEntry.Jerk	 := MoveDynamics.GetJ(Coord_Mcs_A1);
	LogEntry.Vlocity := MoveDynamics.GetV(Coord_Mcs_A1);
	UpdateLog();
	HasRun := TRUE;
END_IF

Execute := THIS^;

//Heartbeat that the method is active
ExecuteWatchdog := ExecuteWatchdog + 1;
END_METHOD

END_FUNCTION_BLOCK

// Mover/TaskClasses/FB_MoveB
FUNCTION_BLOCK FB_MoveB EXTENDS FB_MoverTaskResult
VAR
END_VAR

METHOD Execute : I_PlanarTaskResult
VAR_INPUT
	Position	 : LREAL;
	MoveDynamics : DynamicConstraint_Coordinates;
END_VAR
IF NOT HasRun THEN
	_Done	 := FALSE;
	_Error	 := FALSE;
	_Busy	 := FALSE;
	_ErrorID := 0;
	ipMover.pm.MoveB(_PlanarFb, Position, MoveDynamics);

	//Update mover command log				
	LogEntry.Command := CONCAT('MoveB : ', TO_STRING(Position));
	LogEntry.Accel	 := MoveDynamics.GetA(Coord_Mcs_B1);
	LogEntry.Decel	 := MoveDynamics.GetD(Coord_Mcs_B1);
	LogEntry.Jerk	 := MoveDynamics.GetJ(Coord_Mcs_B1);
	LogEntry.Vlocity := MoveDynamics.GetV(Coord_Mcs_B1);
	UpdateLog();
	HasRun := TRUE;
END_IF

Execute := THIS^;

//Heartbeat that the method is active
ExecuteWatchdog := ExecuteWatchdog + 1;
END_METHOD

END_FUNCTION_BLOCK

// Mover/TaskClasses/FB_MoveToPosition
FUNCTION_BLOCK FB_MoveToPosition EXTENDS FB_MoverTaskResult
VAR
	MoveOptions : ST_MoveToPositionOptions;
	MoverPosition : MoverVector;
	Position	: PositionXYC;
END_VAR

METHOD Execute : I_PlanarTaskResult
VAR_INPUT
	XPosition	 : LREAL;
	YPosition	 : LREAL;
	MoveDynamics : DynamicConstraint_PathXYZ;
END_VAR
IF NOT HasRun THEN
	_Done		  := FALSE;
	_Error		  := FALSE;
	_Busy		  := FALSE;
	_ErrorID	  := 0;
	MoverPosition := ipMover.pm.MCTOPLC.SET.SetPos;
	Position.SetValuesXYC(XPosition, YPosition, MoverPosition.c);
	ipMover.pm.MoveToPosition(_PlanarFb,
							  Position,
							  MoveDynamics,
							  MoveOptions);

	//Update mover command log				
	LogEntry.Command := CONCAT('MoveToPosition : ', CONCAT(CONCAT('X= ', TO_STRING(XPosition)), CONCAT(' Y= ', TO_STRING(YPosition))));
	LogEntry.Accel	 := MoveDynamics.A;
	LogEntry.Decel	 := MoveDynamics.D;
	LogEntry.Jerk	 := MoveDynamics.J;
	LogEntry.Vlocity := MoveDynamics.V;
	UpdateLog();
	HasRun := TRUE;
END_IF

Execute := THIS^;

//Heartbeat that the method is active
ExecuteWatchdog := ExecuteWatchdog + 1;
END_METHOD

END_FUNCTION_BLOCK

// Mover/TaskClasses/FB_MoveZ
FUNCTION_BLOCK FB_MoveZ EXTENDS FB_MoverTaskResult
VAR
END_VAR

METHOD Execute : I_PlanarTaskResult
VAR_INPUT
	Position	 : LREAL;
	MoveDynamics : DynamicConstraint_PathXYZ;
END_VAR
IF NOT HasRun THEN
	_Done	 := FALSE;
	_Error	 := FALSE;
	_Busy	 := FALSE;
	_ErrorID := 0;
	ipMover.pm.MoveZ(_PlanarFb, Position, MoveDynamics);

	//Update mover command log				
	LogEntry.Command := CONCAT('MoveZ : ', TO_STRING(Position));
	LogEntry.Accel	 := MoveDynamics.A;
	LogEntry.Decel	 := MoveDynamics.D;
	LogEntry.Jerk	 := MoveDynamics.J;
	LogEntry.Vlocity := MoveDynamics.V;
	UpdateLog();
	HasRun := TRUE;
END_IF

Execute := THIS^;

//Heartbeat that the method is active
ExecuteWatchdog := ExecuteWatchdog + 1;
END_METHOD

END_FUNCTION_BLOCK

// Mover/TaskClasses/FB_ResetMover
FUNCTION_BLOCK FB_ResetMover EXTENDS FB_MoverTaskResult
VAR
END_VAR

METHOD Execute : I_PlanarTaskResult
IF NOT HasRun THEN
	_Done		:= FALSE;
	_Error		:= FALSE;
	_Busy		:= FALSE;
	_ErrorID	:= 0;
	ipMover.pm.Reset(_PlanarFb);
	HasRun := TRUE;
END_IF

Execute := THIS^;

//Heartbeat that the method is active
ExecuteWatchdog := ExecuteWatchdog + 1;
END_METHOD

END_FUNCTION_BLOCK

// Mover/TaskClasses/FB_Rotate
FUNCTION_BLOCK FB_Rotate EXTENDS FB_MoverTaskResult
VAR
	RotateOptions : ST_MoveCOptions;
END_VAR

METHOD Execute : I_PlanarTaskResult
VAR_INPUT
	Distance	   : LREAL;
	NumberOfTurns  : DINT;
	Direction	   : Tc3_Mc3PlanarMotion.MC_DIRECTION;
	RotateDynamics : DynamicConstraint_Coordinates;
END_VAR
IF NOT HasRun THEN
	_Done						  := FALSE;
	_Error						  := FALSE;
	_Busy						  := FALSE;
	_ErrorID					  := 0;
	RotateOptions.direction		  := Direction;
	RotateOptions.additionalTurns := TO_UDINT(NumberOfTurns);
	ipMover.pm.MoveC(_PlanarFb,
					 Distance,
					 RotateDynamics,
					 RotateOptions);

	//Update mover command log				
	LogEntry.Command := CONCAT('MoveC : ', CONCAT(TO_STRING(Distance), CONCAT(' : Turns ', TO_STRING(NumberOfTurns))));
	LogEntry.Accel	 := RotateDynamics.GetA(Coord_Mcs_C1);
	LogEntry.Decel	 := RotateDynamics.GetD(Coord_Mcs_C1);
	LogEntry.Jerk	 := RotateDynamics.GetJ(Coord_Mcs_C1);
	LogEntry.Vlocity := RotateDynamics.GetV(Coord_Mcs_C1);
	UpdateLog();
	HasRun := TRUE;
END_IF

Execute := THIS^;

//Heartbeat that the method is active
ExecuteWatchdog := ExecuteWatchdog + 1;
END_METHOD

END_FUNCTION_BLOCK

// Mover/TaskClasses/FB_SquareUp
FUNCTION_BLOCK FB_SquareUp EXTENDS FB_MoverTaskResult
VAR
	RotateOptions	: Tc3_Mc3PlanarMotion.ST_MoveCOptions;
	_RotateDynamics : Tc3_Physics.DynamicConstraint_Coordinates;
	_MoveDynamics	: Tc3_Physics.DynamicConstraint_PathXYZ;
	_Distance		: LREAL;
	SquareUp		: BOOL;
END_VAR

METHOD Execute : I_PlanarTaskResult
VAR_INPUT
	Distance	   : LREAL;
	RotateDynamics : Tc3_Physics.DynamicConstraint_Coordinates;
	MoveDynamics   : Tc3_Physics.DynamicConstraint_PathXYZ;
END_VAR
IF NOT HasRun THEN
	_Done			:= FALSE;
	_Error			:= FALSE;
	_Busy			:= FALSE;
	_ErrorID		:= 0;
	_Distance		:= Distance;
	_RotateDynamics := RotateDynamics;
	_MoveDynamics	:= MoveDynamics;
	SquareUp		:= TRUE;
	HasRun			:= TRUE;
END_IF

Execute := THIS^;

//Heartbeat that the method is active
ExecuteWatchdog := ExecuteWatchdog + 1;
END_METHOD

METHOD Update
VAR_INST
	WatchdogCheck : UDINT;
END_VAR
//***Overwriting the update method because this task contains a state machine that must be monitored cyclically.***
_PlanarFb.Update();

//State logic for the task
CASE TaskState OF
	0: // Init
		_Busy := FALSE;
		IF SquareUp THEN
			_Done	  := FALSE;
			_Error	  := FALSE;
			_ErrorID  := 0;
			_Busy	  := TRUE;
			SquareUp  := FALSE;
			TaskState := TaskState + 10;
		END_IF

	10: //Rotate C to closest quarter angle
		RotateOptions.direction		  := Tc3_Mc3PlanarMotion.MC_DIRECTION.mcDirectionShortestWay;
		RotateOptions.additionalTurns := 0;
		ipMover.pm.MoveC(_PlanarFb,
						 _Distance,
						 _RotateDynamics,
						 RotateOptions);

		//Update mover command log				
		LogEntry.Command := CONCAT('MoveC : ', TO_STRING(_Distance));
		LogEntry.Accel	 := _RotateDynamics.GetA(Coord_Mcs_C1);
		LogEntry.Decel	 := _RotateDynamics.GetD(Coord_Mcs_C1);
		LogEntry.Jerk	 := _RotateDynamics.GetJ(Coord_Mcs_C1);
		LogEntry.Vlocity := _RotateDynamics.GetV(Coord_Mcs_C1);
		UpdateLog();
		TaskState := TaskState + 10;

	20: //Watch rotate feedback
		IF _PlanarFb.Done THEN
			TaskState := TaskState + 10;
		ELSIF _PlanarFb.Error THEN
			TaskState := 999;
		END_IF

	30: //Move A Axis to 0
		ipMover.pm.MoveA(_PlanarFb, 0.0, _MoveDynamics);

		//Update mover command log				
		LogEntry.Command := CONCAT('Move A : ', TO_STRING(0.0));
		LogEntry.Accel	 := _MoveDynamics.A;
		LogEntry.Decel	 := _MoveDynamics.D;
		LogEntry.Jerk	 := _MoveDynamics.J;
		LogEntry.Vlocity := _MoveDynamics.V;
		UpdateLog();
		TaskState := TaskState + 10;

	40: //A Axis move feedback
		IF _PlanarFb.Done THEN
			TaskState := TaskState + 10;
		ELSIF _PlanarFb.Error THEN
			TaskState := 999;
		END_IF

	50: //Move B Axis to 0
		ipMover.pm.MoveB(_PlanarFb, 0.0, _MoveDynamics);

		//Update mover command log				
		LogEntry.Command := CONCAT('Move B : ', TO_STRING(0.0));
		LogEntry.Accel	 := _MoveDynamics.A;
		LogEntry.Decel	 := _MoveDynamics.D;
		LogEntry.Jerk	 := _MoveDynamics.J;
		LogEntry.Vlocity := _MoveDynamics.V;
		UpdateLog();
		TaskState := TaskState + 10;

	60: //A Axis move feedback
		IF _PlanarFb.Done THEN
			TaskState := TaskState + 10;
		ELSIF _PlanarFb.Error THEN
			TaskState := 999;
		END_IF

	70: //Task Complete
		_Done	  := TRUE;
		TaskState := 0;

	999: //Task Error
		_Error				:= TRUE;
		_ErrorID			:= _PlanarFb.ErrorId;
		_BlockingObjectInfo := _PlanarFb.objectInfo;
		TaskState			:= 0;
END_CASE

RT_ADSWarn(CLK := _PlanarFb.Error);
IF RT_ADSWarn.Q THEN
	ADSLOGSTR(ADSLOG_MSGTYPE_WARN, CONCAT('Mover ', ipMover.MoverBTN), CONCAT(_TaskName, CONCAT('Error ', TO_STRING(_PlanarFb.ErrorId))));
END_IF

IF ExecuteWatchdog <> WatchdogCheck THEN
	WatchdogCheck := ExecuteWatchdog;
ELSE
	HasRun			:= FALSE;
	ExecuteWatchdog := 0;
END_IF
END_METHOD

END_FUNCTION_BLOCK

// Mover/TaskClasses/FB_TrackMove
FUNCTION_BLOCK FB_TrackMove EXTENDS FB_MoverTaskResult
VAR
	DynMove			   : DynamicConstraint_PathXY;
	MoveOnTrackOptions : ST_MoveOnTrackOptions;
	MoverSetPos		   : MoverVector;
	OnTrackPos		   : LREAL;
END_VAR

METHOD Execute : I_PlanarTaskResult
VAR_INPUT
	Position	 : LREAL;
	Gap			 : LREAL;
	TrackSegment : I_XPlanarTrack;
	MoveDynamics : DynamicConstraint_PathXY;
END_VAR
IF NOT HasRun AND (ipMover.Status.CommandMode = MC_Planar_Mover_Command_Mode.OnTrack OR ipMover.Status.CommandMode = MC_Planar_Mover_Command_Mode.CRotationOnTrack) THEN
	_Done		:= FALSE;
	_Error		:= FALSE;
	_Busy		:= FALSE;
	_ErrorID	:= 0;
	MoveOnTrackOptions.gap		 := Gap;
	MoveOnTrackOptions.direction := MC_Direction.mcDirectionPositive;
	ipMover.pm.MoveOnTrack(_PlanarFb,
					  TrackSegment.pm,
					  Position,
					  MoveDynamics,
					  MoveOnTrackOptions);

	//Update mover command log				
	LogEntry.Command := CONCAT('MoveOnTrack : ', CONCAT(CONCAT('ID : ', TO_STRING(TrackSegment.Index)), CONCAT(' Pos ', TO_STRING(Position))));
	LogEntry.Accel	 := MoveDynamics.A;
	LogEntry.Decel	 := MoveDynamics.D;
	LogEntry.Jerk	 := MoveDynamics.J;
	LogEntry.Vlocity := MoveDynamics.V;
	UpdateLog();
	HasRun := TRUE;
END_IF

Execute := THIS^;

//Heartbeat that the method is active
ExecuteWatchdog := ExecuteWatchdog + 1;
END_METHOD

END_FUNCTION_BLOCK

// Mover/TaskClasses/FB_TrackMoveXY
FUNCTION_BLOCK FB_TrackMoveXY EXTENDS FB_MoverTaskResult
VAR
	DynMove			   : DynamicConstraint_PathXY;
	MoveOnTrackOptions : ST_MoveOnTrackOptions;
END_VAR

METHOD Execute : I_PlanarTaskResult
VAR_INPUT
	PositionX	 : LREAL;
	PositionY	 : LREAL;
	Gap			 : LREAL;
	TrackSegment : I_XPlanarTrack;
	MoveDynamics : DynamicConstraint_PathXY;
END_VAR

VAR_INST
	Position		: PositionXYC;
	SetPosition		: MoverVector;
	OnTrackPosition : LREAL;
END_VAR
IF NOT HasRun AND (ipMover.Status.CommandMode = MC_Planar_Mover_Command_Mode.OnTrack OR ipMover.Status.CommandMode = MC_Planar_Mover_Command_Mode.CRotationOnTrack) THEN
	_Done		:= FALSE;
	_Error		:= FALSE;
	_Busy		:= FALSE;
	_ErrorID	:= 0;
	SetPosition := ipMover.pm.MCTOPLC.SET.SetPos;
	Position.SetValuesXY(PositionX, PositionY);
	MoveOnTrackOptions.gap		 := Gap;
	MoveOnTrackOptions.direction := Tc3_Mc3PlanarMotion.MC_Direction.mcDirectionPositive;
	OnTrackPosition				 := TrackSegment.GetTrackPositionAt(Position);
	ipMover.pm.MoveOnTrack(_PlanarFb,
					  TrackSegment.pm,
					  OnTrackPosition,
					  MoveDynamics,
					  MoveOnTrackOptions);

	//Update mover command log				
	LogEntry.Command := CONCAT('MoveOnTrack : ', CONCAT(CONCAT('ID : ', TO_STRING(TrackSegment.Index)), CONCAT(' Pos ', TO_STRING(OnTrackPosition))));
	LogEntry.Accel	 := MoveDynamics.A;
	LogEntry.Decel	 := MoveDynamics.D;
	LogEntry.Jerk	 := MoveDynamics.J;
	LogEntry.Vlocity := MoveDynamics.V;
	UpdateLog();
	HasRun := TRUE;
END_IF

Execute := THIS^;

//Heartbeat that the method is active
ExecuteWatchdog := ExecuteWatchdog + 1;
END_METHOD

END_FUNCTION_BLOCK

// Mover/FB_XPlanarMover
FUNCTION_BLOCK FB_XPlanarMover EXTENDS FB_CyclicFB IMPLEMENTS I_XPlanarMover, I_MoveCommands, I_MoveDynamics
VAR
	_Mover		: Tc3_MC3PlanarMotion.MC_PlanarMover;
	_ObjectInfo : Tc3_Mc3PlanarMotion.PlanarObjectInfo;
	_std		: CDT_MCTOPLC_PLANAR_MOVER_STD;

	//Command Log
	_CommandLog : ARRAY[0..SystemParameters.MAX_LOG_COUNT] OF ST_CommandLog;

	//Mover Task Declarations
	EnableMover			 : FB_Enable		   := (Mover := THIS^, TaskName := 'Enable');
	DisableMover		 : FB_Disable		   := (Mover := THIS^, TaskName := 'Disable');
	HaltMover			 : FB_Halt			   := (Mover := THIS^, TaskName := 'Halt');
	JoinMoverToTrack	 : FB_JoinTrack		   := (Mover := THIS^, TaskName := 'JoinTrack');
	JoinToClosestTrack	 : FB_JoinClosestTrack := (Mover := THIS^, TaskName := 'JoinClosestTrack');
	LeaveMoverFromTrack	 : FB_LeaveTrack	   := (Mover := THIS^, TaskName := 'LeaveTrack');
	ResetMover			 : FB_ResetMover	   := (Mover := THIS^, TaskName := 'Reset');
	MoveOnTrackXY		 : FB_TrackMoveXY	   := (Mover := THIS^, TaskName := 'MoveOnTrack');
	MoveOnTrack			 : FB_TrackMove		   := (Mover := THIS^, TaskName := 'MoveOnTrack');
	RotateMover			 : FB_Rotate		   := (Mover := THIS^, TaskName := 'Rotate');
	ZMove				 : FB_MoveZ			   := (Mover := THIS^, TaskName := 'MoveZ');
	AMove				 : FB_MoveA			   := (Mover := THIS^, TaskName := 'MoveA');
	BMove				 : FB_MoveB			   := (Mover := THIS^, TaskName := 'MoveB');
	MoveToPosition		 : FB_MoveToPosition   := (Mover := THIS^, TaskName := 'MoveToPosition');
	AddMoverToGroup		 : FB_AddToGroup	   := (Mover := THIS^, TaskName := 'AddToGroup');
	SquareMover			 : FB_SquareUp		   := (Mover := THIS^, TaskName := 'SquareUp');
	InvalidCommandResult : FB_ResultBase	   := (Busy := FALSE, Error := TRUE, ErrorID := 9999);

	//Internal Vars
	_MoveDynamics		 : ST_MoveDynamics;
	_RotateDynamics		 : ST_MoveDynamics;
	_TiltDynamics		 : ST_MoveDynamics;
	_DynMove			 : Tc3_Physics.DynamicConstraint_PathXYZ;
	_DynRotate			 : Tc3_Physics.DynamicConstraint_Coordinates;
	_DynTrackMove		 : Tc3_Physics.DynamicConstraint_PathXY;
	_DynHalt			 : Tc3_Physics.DynamicConstraint_PathXYZ;
	_Gap				 : LREAL;
	_MoverIndex			 : UDINT;
	_TrackId			 : UDINT;
	_MoverBTN			 : STRING;
	_IdentifiedBTN		 : STRING;
	_MoverType			 : XPlanarMoverType;
	_InStation			 : BOOL;
	ipDestination		 : I_XPlanarStation;
	ipMoverTcIo			 : I_TcIoXPlanarMover;
	_ModuloPosC			 : LREAL;
	TypeIsRead			 : BOOL;
	ClosestSquarePos	 : LREAL;
	_MoverActPos		 : MoverVector;
	_ClosestQuarterAngle : LREAL;
	_AtRotationPosition	 : BOOL;
	UpdateMoveDynamics	 : BOOL;
	UpdateRotateDynamics : BOOL;
	UpdateTiltDynamics	 : BOOL;
END_VAR

(*
HaltDynamics.Mode				  := E_HaltDynamicsMode.AxisX_AxisY_CoordinatedOnPath;
HaltDynamics.PathXY.fVelocity     := 500.0;
HaltDynamics.PathXY.fAcceleration := 10000.0;
HaltDynamics.PathXY.fDeceleration := 10000.0;
HaltDynamics.PathXY.fJerk         := 100000.0;
HaltDynamics.AxisX.fVelocity      := 500.0;
HaltDynamics.AxisX.fAcceleration  := 10000.0;
HaltDynamics.AxisX.fDeceleration  := 10000.0;
HaltDynamics.AxisX.fJerk          := 100000.0;
HaltDynamics.AxisY.fVelocity      := 500.0;
HaltDynamics.AxisY.fAcceleration  := 10000.0;
HaltDynamics.AxisY.fDeceleration  := 10000.0;
HaltDynamics.AxisY.fJerk          := 100000.0;
HaltDynamics.AxisZ.fVelocity      := 500.0;
HaltDynamics.AxisZ.fAcceleration  := 10000.0;
HaltDynamics.AxisZ.fDeceleration  := 10000.0;
HaltDynamics.AxisZ.fJerk          := 100000.0;
HaltDynamics.AxisA.fVelocity      := 10.0;
HaltDynamics.AxisA.fAcceleration  := 100.0;
HaltDynamics.AxisA.fDeceleration  := 100.0;
HaltDynamics.AxisA.fJerk          := 100.0;
HaltDynamics.AxisB.fVelocity      := 10.0;
HaltDynamics.AxisB.fAcceleration  := 100.0;
HaltDynamics.AxisB.fDeceleration  := 100.0;
HaltDynamics.AxisB.fJerk          := 100.0;
HaltDynamics.AxisC.fVelocity      := 36.0;
HaltDynamics.AxisC.fAcceleration  := 360.0;
HaltDynamics.AxisC.fDeceleration  := 360.0;
HaltDynamics.AxisC.fJerk          := 360.0;
*)

{attribute 'TcRpcEnable'}
METHOD FreeMove : I_PlanarTaskResult
VAR_INPUT
	XPosition : LREAL;
	YPosition : LREAL;
END_VAR

VAR_INST
	Position : PositionXYC;
END_VAR
FreeMove := MoveToPosition.Execute(XPosition, YPosition, _DynMove);
END_METHOD

{attribute 'TcRpcEnable'}
METHOD JoinClosestTrack : I_PlanarTaskResult
VAR_INPUT
	UseOrientation : BOOL;
END_VAR
JoinClosestTrack := JoinToClosestTrack.Execute(UseOrientation, _DynMove);
END_METHOD

{attribute 'TcRpcEnable'}
METHOD JoinTrack : I_PlanarTaskResult
VAR_INPUT
	ipTrack		   : I_XPlanarTrack;
	UseOrientation : BOOL;
END_VAR
JoinTrack := JoinMoverToTrack.Execute(ipTrack, UseOrientation, _DynMove);
END_METHOD

{attribute 'TcRpcEnable'}
METHOD LeaveTrack : I_PlanarTaskResult
VAR_INPUT
	DestinationX   : LREAL;
	DestinationY   : LREAL;
	UseOrientation : BOOL;
END_VAR

VAR_INST
	Destination : PositionXYC;
END_VAR
LeaveTrack := LeaveMoverFromTrack.Execute(DestinationX,
										  DestinationY,
										  UseOrientation,
										  _DynMove);
END_METHOD

{attribute 'TcRpcEnable'}
METHOD Rotate : I_PlanarTaskResult
VAR_INPUT
	Position		: LREAL;
	AdditionalTurns : DINT;
END_VAR

VAR
	Direction : Tc3_Mc3PlanarMotion.MC_DIRECTION;
END_VAR
IF AdditionalTurns < 0 OR Position < 0 THEN
	Direction := Tc3_Mc3PlanarMotion.MC_DIRECTION.mcDirectionNegative;
ELSIF Position = 0 AND AdditionalTurns = 0 THEN
	Direction := Tc3_Mc3PlanarMotion.MC_DIRECTION.mcDirectionShortestWay;
ELSE
	Direction := Tc3_Mc3PlanarMotion.MC_DIRECTION.mcDirectionPositive;
END_IF

IF _AtRotationPosition OR ((Position >= -10 OR Position <= 10) AND AdditionalTurns = 0) THEN
	Rotate := RotateMover.Execute(ABS(Position),
								  ABS(AdditionalTurns),
								  Direction,
								  _DynRotate);
ELSE
	Rotate := InvalidCommandResult;
END_IF
END_METHOD

{attribute 'TcRpcEnable'}
METHOD SendToStation : I_PlanarTaskResult
VAR_INPUT
	Destination : I_XPlanarStation;
END_VAR

VAR_INST
	CorrectedPos : PositionXYC;
	OnTrackPos	 : LREAL;
END_VAR
ipDestination := Destination; //Update the destination field of the mover
IF _Mover.MCTOPLC.STD.CommandMode = MC_PLANAR_MOVER_COMMAND_MODE.OnTrack THEN
	IF Destination.TrackID <> 0 THEN
		SendToStation := MoveOnTrackXY.Execute(Destination.Position.x,
											 Destination.Position.y,
											 _Gap,
											 ip.Tracks[Destination.TrackID],
											 _DynTrackMove);

		IF SystemParameters.EnableCommandTracing THEN
			THIS^.Trace(CONCAT(CONCAT('Mover ', TO_STRING(_MoverIndex)), CONCAT(', ', CONCAT('TrackMoveToStation ', TO_STRING(Destination.ID)))));
		END_IF
	ELSE
		SendToStation := InvalidCommandResult;
	END_IF
ELSIF _Mover.MCTOPLC.STD.CommandMode = MC_PLANAR_MOVER_COMMAND_MODE.FreeMovement THEN
	CorrectedPos.SetValuesXYC(Destination.Position.x, Destination.Position.y, _MoverActPos.c);
	SendToStation := MoveToPosition.Execute(Destination.Position.x, Destination.Position.y, _DynMove);
	IF SystemParameters.EnableCommandTracing THEN
		THIS^.Trace(CONCAT(CONCAT('Mover ', TO_STRING(_MoverIndex)), CONCAT(', ', CONCAT('FreeMoveToStation ', TO_STRING(Destination.ID)))));
	END_IF
ELSE
	SendToStation := InvalidCommandResult;
END_IF
END_METHOD

{attribute 'TcRpcEnable'}
METHOD SquareUp : I_PlanarTaskResult
VAR_INST
	Result		 : FB_ResultBase;
END_VAR
SquareUp := SquareMover.Execute(_ClosestQuarterAngle, _DynRotate, _DynMove);
END_METHOD

METHOD TiltA : I_PlanarTaskResult
VAR_INPUT
	Position : LREAL;
END_VAR
TiltA := AMove.Execute(Position, _DynRotate);
END_METHOD

METHOD TiltB : I_PlanarTaskResult
VAR_INPUT
	Position : LREAL;
END_VAR
TiltB := BMove.Execute(Position, _DynRotate);
END_METHOD

{attribute 'TcRpcEnable'}
METHOD TrackMove : I_PlanarTaskResult
VAR_INPUT
	Position : LREAL;
	Gap		  : LREAL;
	Track	  : I_XPlanarTrack;
	Direction : Tc3_Mc3PlanarMotion.MC_DIRECTION;
END_VAR

VAR
	WorkingGap : LREAL;
END_VAR
IF Gap > 0 THEN
	WorkingGap := Gap;
ELSE
	WorkingGap := _Gap;
END_IF

TrackMove := MoveOnTrack.Execute(Position,
								 WorkingGap,
								 Track,
								 _DynTrackMove);
END_METHOD

{attribute 'TcRpcEnable'}
METHOD TrackMoveXY : I_PlanarTaskResult
VAR_INPUT
	XPosition : LREAL;
	YPosition : LREAL;
	Gap		  : LREAL;
	Track	  : I_XPlanarTrack;
	Direction : Tc3_Mc3PlanarMotion.MC_DIRECTION;
END_VAR

VAR
	WorkingGap : LREAL;
END_VAR

VAR_INST
	Position   : PositionXYC;
	OnTrackPos : LREAL;
END_VAR
IF Gap > 0 THEN
	WorkingGap := Gap;
ELSE
	WorkingGap := _Gap;
END_IF

TrackMoveXY := MoveOnTrackXY.Execute(XPosition,
								   YPosition,
								   WorkingGap,
								   Track,
								   _DynTrackMove);
END_METHOD

{attribute 'TcRpcEnable'}
METHOD VerticalMove : I_PlanarTaskResult
VAR_INPUT
	Position : LREAL;
END_VAR
VerticalMove := ZMove.Execute(Position, _DynMove);
END_METHOD

PROPERTY Movement : REFERENCE TO ST_MoveDynamics
GET
Movement REF= _MoveDynamics;
UpdateMoveDynamics := TRUE;
END_GET
END_PROPERTY

PROPERTY Rotation : REFERENCE TO ST_MoveDynamics
GET
Rotation REF= _RotateDynamics;
UpdateRotateDynamics := true;
END_GET
END_PROPERTY

PROPERTY Tilt : REFERENCE TO ST_MoveDynamics
GET
Tilt REF= _TiltDynamics;
UpdateTiltDynamics := TRUE;
END_GET
END_PROPERTY

PROPERTY ActualPosition : REFERENCE TO MoverVector
GET
ActualPosition ref= _MoverActPos;
END_GET
END_PROPERTY

METHOD AddToGroup : I_PlanarTaskResult
VAR_INPUT
	PlanarGroup : REFERENCE TO MC_PlanarGroup;
END_VAR
AddToGroup := AddMoverToGroup.Execute(PlanarGroup);
END_METHOD

PROPERTY CommandLog : REFERENCE TO ARRAY [0..SystemParameters.MAX_LOG_COUNT] of ST_CommandLog
GET
CommandLog ref= _CommandLog;
END_GET
END_PROPERTY

PROPERTY Destination : I_XPlanarStation
GET
Destination := ipDestination;
END_GET
SET
ipDestination := Destination;
END_SET
END_PROPERTY

{attribute 'TcRpcEnable'}
METHOD Disable : I_PlanarTaskResult
Disable := DisableMover.Execute();
END_METHOD

PROPERTY Dynamics : I_MoveDynamics
GET
Dynamics := THIS^;
END_GET
END_PROPERTY

{attribute 'TcRpcEnable'}
METHOD Enable : I_PlanarTaskResult
Enable := EnableMover.Execute();
END_METHOD

PROPERTY Gap : LREAL
GET
Gap := _Gap;
END_GET
SET
_Gap := Gap;
END_SET
END_PROPERTY

METHOD Halt : I_PlanarTaskResult
Halt := HaltMover.Execute(_DynHalt);
END_METHOD

PROPERTY IdentifiedBTN : STRING
GET
IF ipMoverTcIo <> 0 THEN
	_IdentifiedBTN := ipMoverTcIo.GetIdentifiedMoverBtn();
END_IF

IdentifiedBTN := _IdentifiedBTN;
END_GET
END_PROPERTY

PROPERTY InStation : BOOL
GET
InStation := _InStation;
END_GET
SET
_InStation := InStation;
END_SET
END_PROPERTY

PROPERTY MoveCommand : I_MoveCommands
GET
MoveCommand := THIS^;
END_GET
END_PROPERTY

PROPERTY MoverBTN : STRING
GET
IF _MoverBTN <> '' THEN
	IF ipMoverTcIo <> 0 THEN
		_MoverBTN := ipMoverTcIo.GetBtn();
	END_IF
END_IF

MoverBTN := _MoverBTN;
END_GET
END_PROPERTY

PROPERTY MoverIndex : UDINT
GET
MoverIndex := _MoverIndex;
END_GET
SET
_MoverIndex := MoverIndex;
END_SET
END_PROPERTY

PROPERTY MoverType : XPlanarMoverType
GET
MoverType := _MoverType;
END_GET
SET
_MoverType := MoverType;
END_SET
END_PROPERTY

PROPERTY pm : REFERENCE TO MC_PlanarMover
GET
pm ref= _Mover;
END_GET
END_PROPERTY

//! @summary Clears error flags and error IDs for this component
{attribute 'TcRpcEnable'}
METHOD PUBLIC Reset : I_PlanarTaskResult
Reset := ResetMover.Execute();
END_METHOD

PROPERTY Status : REFERENCE TO CDT_MCTOPLC_PLANAR_MOVER_STD
GET
Status ref= _Std;
END_GET
END_PROPERTY

PROPERTY Utility : I_TcIoXPlanarMover
GET
IF ipMoverTcIo <> 0 THEN
	Utility := ipMoverTcIo;
END_IF
END_GET
SET
ipMoverTcIo := Utility;
END_SET
END_PROPERTY

//! @summary This method serves as the entry point for all underlying FB logic
METHOD PUBLIC CyclicLogic
//! @description This method should be called cyclically by descendant function blocks by invoking <c>SUPER^.CyclicLogic()</c>.  Alternatively, the contents of this method could be reimplemented entirely in which case a call to this method would not be necessary.
VAR
	Result : BOOL;
END_VAR

VAR_INST
	MoverSetPos	 : MoverVector;
	ModXPos		 : LREAL;
	ModXPosRound : LREAL;
	ModYPos		 : LREAL;
	ModYPosRound : LREAL;
	FracX		 : LREAL;
	FracY		 : LREAL;
END_VAR
//Keep Task command feedbacks up to date
EnableMover.Update();
DisableMover.Update();
HaltMover.Update();
JoinMoverToTrack.Update();
LeaveMoverFromTrack.Update();
ResetMover.Update();
MoveOnTrackXY.Update();
MoveOnTrack.Update();
RotateMover.Update();
ZMove.Update();
AMove.Update();
BMove.Update();
MoveToPosition.Update();
AddMoverToGroup.Update();
JoinToClosestTrack.Update();
SquareMover.Update();

//Update Mover MC Info
_std	 := _Mover.MCTOPLC.STD;
_Busy	 := _std.Busy.busyMover;
_Error	 := _Mover.Error;
_ErrorID := _Mover.ErrorId;

//Calculate Mover Closest Quarter Angle
_MoverActPos := _Mover.MCTOPLC.ACT.ActPos;
_ModuloPosC	 := LMOD(_MoverActPos.c, 360.0);
IF _ModuloPosC < 315.0 AND _ModuloPosC > 225.0 THEN
	_ClosestQuarterAngle := 270.0;
ELSIF _ModuloPosC < 225.0 AND _ModuloPosC > 135.0 THEN
	_ClosestQuarterAngle := 180.0;
ELSIF _ModuloPosC < 135.0 AND _ModuloPosC > 45.0 THEN
	_ClosestQuarterAngle := 90.0;
ELSE
	_ClosestQuarterAngle := 0.0;
END_IF

//Determine if Mover is at a valid rotation position
MoverSetPos			:= _Mover.MCTOPLC.SET.SetPos;
ModXPos				:= LMOD(MoverSetPos.x, 120.0);
ModXPosRound		:= TO_LREAL(TO_DINT(ModXPos * (2 * 10))) / (2 * 10); //Round the Modulo position to 2 decimal places
FracX				:= FRAC(ModXPosRound);
ModYPos				:= LMOD(MoverSetPos.y, 120.0);
ModYPosRound		:= TO_LREAL(TO_DINT(ModYPos * (2 * 10))) / (2 * 10); //Round the Modulo position to 2 decimal places
FracY				:= FRAC(ModYPosRound);
_AtRotationPosition := (MoverSetPos.x >= 120 AND FracX = 0) AND (MoverSetPos.y >= 120 AND FracY = 0);

//Monitor Changes in move dynamic settings
IF UpdateMoveDynamics THEN
	_DynMove.SetValuesVADJ(_MoveDynamics.Velocity,
						   _MoveDynamics.Accel,
						   _MoveDynamics.Decel,
						   _MoveDynamics.Jerk);

	_DynTrackMove.SetValuesVADJ(_MoveDynamics.Velocity,
								_MoveDynamics.Accel,
								_MoveDynamics.Decel,
								_MoveDynamics.Jerk);

	UpdateMoveDynamics := FALSE;
END_IF

IF UpdateRotateDynamics THEN
	_DynRotate.SetLimit(Coord_Mcs_C1,
						_RotateDynamics.Velocity,
						_RotateDynamics.Accel,
						_RotateDynamics.Decel,
						_RotateDynamics.Jerk);

	UpdateRotateDynamics := FALSE;
END_IF

IF UpdateTiltDynamics THEN
	_DynRotate.SetLimit(Coord_Mcs_A1,
						_TiltDynamics.Velocity,
						_TiltDynamics.Accel,
						_TiltDynamics.Decel,
						_TiltDynamics.Jerk);

	_DynRotate.SetLimit(Coord_Mcs_B1,
						_TiltDynamics.Velocity,
						_TiltDynamics.Accel,
						_TiltDynamics.Decel,
						_TiltDynamics.Jerk);

	UpdateTiltDynamics := FALSE;
END_IF

//Update Mover Position for HMI
IF _MoverIndex > 0 AND _MoverIndex <= SystemParameters.MOVER_COUNT THEN
	XPlanarHMI.MoverPositions[_MoverIndex] := _MoverActPos;
END_IF
END_METHOD

END_FUNCTION_BLOCK

// Part/Tasks/FB_AllowEnable
FUNCTION_BLOCK FB_AllowEnable EXTENDS FB_PartTaskResult
VAR
END_VAR

METHOD Execute : I_PlanarTaskResult
VAR_INPUT
END_VAR
IF NOT HasRun THEN
	_Done	 := FALSE;
	_Error	 := FALSE;
	_Busy	 := FALSE;
	_ErrorID := 0;
	ipPart.pm.AllowEnable(_PlanarFb);
	HasRun := TRUE;
END_IF

Execute := THIS^;
END_METHOD

END_FUNCTION_BLOCK

// XPlanarResultClasses/FB_PartTaskResult
FUNCTION_BLOCK FB_PartTaskResult EXTENDS FB_PlanarFeedbackResult
VAR
	ipPart : I_XplanarPart;
END_VAR

PROPERTY Part : I_XPlanarPart
SET
ipPart := Part;
END_SET
END_PROPERTY

END_FUNCTION_BLOCK

// Part/I_XPlanarPart
INTERFACE I_XPlanarPart EXTENDS I_BaseFB

METHOD ForceDisable : I_PlanarTaskResult
END_METHOD

PROPERTY ObjectID : OTCID
GET
END_GET
END_PROPERTY

PROPERTY pm : REFERENCE TO MC_PlanarPart
GET
END_GET
END_PROPERTY

METHOD Reset : I_PlanarTaskResult
VAR_INPUT
END_VAR
END_METHOD

METHOD SetAllowEnable : I_PlanarTaskResult
END_METHOD

PROPERTY State : REFERENCE TO MC_PLANAR_STATE
GET
END_GET
END_PROPERTY

END_INTERFACE

// Part/Tasks/FB_ForceDisable
FUNCTION_BLOCK FB_ForceDisable EXTENDS FB_PartTaskResult
VAR
END_VAR

METHOD Execute : I_PlanarTaskResult
VAR_INPUT
END_VAR
IF NOT HasRun THEN
	_Done	 := FALSE;
	_Error	 := FALSE;
	_Busy	 := FALSE;
	_ErrorID := 0;
	ipPart.pm.ForceDisable(_PlanarFb);
	HasRun := TRUE;
END_IF

Execute := THIS^;
END_METHOD

END_FUNCTION_BLOCK

// Part/Tasks/FB_Initialize
FUNCTION_BLOCK FB_Initialize EXTENDS FB_PartTaskResult
VAR
END_VAR

METHOD Execute : I_PlanarTaskResult
VAR_INPUT
	OID : OTCID;
END_VAR
IF NOT HasRun THEN
	ipPart.pm.Initialize(_PlanarFb, OID, XPlanar.Environment);
	HasRun := TRUE;
END_IF

Execute := THIS^;
END_METHOD

END_FUNCTION_BLOCK

// Part/Tasks/FB_ResetPart
FUNCTION_BLOCK FB_ResetPart EXTENDS FB_PartTaskResult
VAR
END_VAR

METHOD Execute : I_PlanarTaskResult
VAR_INPUT
END_VAR
IF NOT HasRun THEN
	_Done	 := FALSE;
	_Error	 := FALSE;
	_Busy	 := FALSE;
	_ErrorID := 0;
	ipPart.pm.Reset(_PlanarFb);
	HasRun := TRUE;
END_IF

Execute := THIS^;
END_METHOD

END_FUNCTION_BLOCK

// Part/FB_XPlanarPart
FUNCTION_BLOCK FB_XPlanarPart EXTENDS FB_CyclicFB IMPLEMENTS I_XPlanarPart
VAR
	PlanarPart			 : MC_PlanarPart;
	_ObjectID			 : OTCID;
	InitPart			 : FB_Initialize   := (Part := THIS^);
	AllowPartEnable		 : FB_AllowEnable  := (Part := THIS^);
	ForcePartDisable	 : FB_ForceDisable := (Part := THIS^);
	ResetPart			 : FB_ResetPart	   := (Part := THIS^);
	InvalidCommandResult : FB_ResultBase   := (Busy := FALSE, Error := TRUE, ErrorID := 9999);
END_VAR

METHOD PUBLIC CyclicLogic
VAR_INPUT
END_VAR
InitPart.Update();
AllowPartEnable.Update();
ForcePartDisable.Update();
ResetPart.Update();
END_METHOD

METHOD ForceDisable : I_PlanarTaskResult
ForceDisable := ForcePartDisable.Execute();
END_METHOD

METHOD Initialize : I_PlanarTaskResult
VAR_INPUT
END_VAR
IF _ObjectID <> 0 THEN
	Initialize := InitPart.Execute(_ObjectID);
ELSE
	Initialize := InvalidCommandResult;
END_IF
END_METHOD

PROPERTY ObjectID : OTCID
GET
ObjectID := _ObjectID;
END_GET
SET
_ObjectID := ObjectID;
END_SET
END_PROPERTY

PROPERTY pm : REFERENCE TO MC_PlanarPart
GET
pm  ref= PlanarPart;
END_GET
END_PROPERTY

METHOD Reset : I_PlanarTaskResult
VAR_INPUT
END_VAR
Reset := ResetPart.Execute();
END_METHOD

METHOD SetAllowEnable : I_PlanarTaskResult
SetAllowEnable := AllowPartEnable.Execute();
END_METHOD

PROPERTY State : REFERENCE TO MC_PLANAR_STATE
GET
State := PlanarPart.State;
END_GET
END_PROPERTY

END_FUNCTION_BLOCK

// Project Information/F_GetCompany
// This function has been automatically generated from the project information.
{attribute 'signature_flag' := '1073741824'}
{attribute 'TcGenerated'}
{attribute 'no-analysis'}
FUNCTION F_GetCompany : WSTRING
VAR_INPUT
	
END_VAR

F_GetCompany := "Beckhoff Automation LLC";

END_FUNCTION

// Project Information/F_GetTitle
// This function has been automatically generated from the project information.
{attribute 'signature_flag' := '1073741824'}
{attribute 'TcGenerated'}
{attribute 'no-analysis'}
FUNCTION F_GetTitle : WSTRING
VAR_INPUT
	
END_VAR

F_GetTitle := "XPlanarApplication";

END_FUNCTION

// Project Information/F_GetVersion
// This function has been automatically generated from the project information.
{attribute 'signature_flag' := '1073741824'}
{attribute 'TcGenerated'}
{attribute 'no-analysis'}
FUNCTION F_GetVersion : ST_LibVersion
VAR_INPUT
	
END_VAR

F_GetVersion.iMajor := 1;
F_GetVersion.iMinor := 0;
F_GetVersion.iBuild := 1;
F_GetVersion.iRevision := 0;
F_GetVersion.sVersion := '1.0.1';
F_GetVersion.nFlags := 1;

END_FUNCTION

// Station/FB_XPlanarStationBase
FUNCTION_BLOCK FB_XPlanarStationBase EXTENDS FB_ComponentBase IMPLEMENTS I_XPlanarStation
VAR
	_Position			 : PositionXYC; //Position of center of the zone
	ipCurrentMover		 : I_XPlanarMover;
	_MoverQueue			 : FB_MoverQueue;
	_NumMoversRequired	 : UDINT := 1;
	_ID					 : UDINT;
	_Size				 : Position2D_LREAL := (x := 120, y := 120); //Size of zone in mm
	_HasMover			 : BOOL;
	_Occupied			 : BOOL;
	ipTrackID			 : UDINT;		 //ID of track that zone resides on
	_CanReleaseMover	 : BOOL := TRUE; //Set to 0 if station area is blocked
	_StationReady AT %Q* : BOOL;
	ipNextStation		 : I_XPlanarStation;
	_AllowQueing		 : BOOL := TRUE;
	_StationComplete	 : BOOL;
	_StationType		 : E_StationType := E_StationType.Process;
	ipMovers			 : REFERENCE TO ARRAY[1..SystemParameters.MOVER_COUNT] OF I_XPlanarMover;
	PrepState			 : UDINT;
	StationState		 : E_XplanarStationState;
END_VAR

PROPERTY AllowQueing : BOOL
GET
AllowQueing := _AllowQueing;
END_GET
SET
_AllowQueing := AllowQueing;
END_SET
END_PROPERTY

PROPERTY CanReleaseMover : BOOL
SET
_CanReleaseMover := CanReleaseMover;
END_SET
END_PROPERTY

PROPERTY CurrentMover : I_XPlanarMover
GET
IF ipCurrentMover <> 0 THEN
	CurrentMover := ipCurrentMover;
END_IF
END_GET
END_PROPERTY

PROPERTY Error : BOOL
GET
Error := _Error;
END_GET
END_PROPERTY

METHOD Execute
VAR_INST
	i			  : UDINT := 1;
	CommandResult : I_PlanarTaskResult;
END_VAR
WatchForMover();
IF ipCurrentMover <> 0 THEN
	CASE StationState OF
		E_XplanarStationState.StationIdle: //Wait for mover to arrive in position
			IF _HasMover AND _StationReady AND NOT _StationComplete THEN
				IF ipCurrentMover <> 0 THEN
					IF (ipTrackID <> 0 AND (ipCurrentMover.Status.CommandMode = MC_PLANAR_MOVER_COMMAND_MODE.OnTrack OR ipCurrentMover.Status.CommandMode = MC_PLANAR_MOVER_COMMAND_MODE.CRotationOnTrack)) OR (ipTrackID = 0 AND (ipCurrentMover.Status.CommandMode = MC_PLANAR_MOVER_COMMAND_MODE.FreeMovement OR ipCurrentMover.Status.CommandMode = MC_PLANAR_MOVER_COMMAND_MODE.CRotationFreeMovement))
						THEN
						StationState := E_XplanarStationState.ProcessMover;
					END_IF
				END_IF
			END_IF

		E_XplanarStationState.ProcessMover: //Perform the desired processes with the mover
			IF _StationComplete THEN
				IF _StationType = E_StationType.MultiMover THEN
					i			 := 1;
					StationState := E_XPlanarStationState.SendQueue;
				ELSE
					StationState := E_XplanarStationState.SquareUpMover;
				END_IF
			END_IF

		E_XplanarStationState.SquareUpMover: //Check mover for angle that allows X/Y Movement
			IF (ipCurrentMover.Status.CommandMode = MC_PLANAR_MOVER_COMMAND_MODE.CRotationOnTrack) OR (ipCurrentMover.Status.CommandMode = MC_PLANAR_MOVER_COMMAND_MODE.CRotationFreeMovement) THEN
				CommandResult := ipCurrentMover.MoveCommand.SquareUp();
				IF CommandResult.Done THEN
					StationState := E_XplanarStationState.SendMoverAway;
				END_IF
			ELSE
				StationState := E_XplanarStationState.SendMoverAway;
			END_IF

		E_XplanarStationState.SendMoverAway: //Send the current lead mover away
			IF ipNextStation <> 0 AND _CanReleaseMover THEN
				IF (NOT ipNextStation.HasMover OR ipNextStation.AllowQueing) THEN
					CommandResult := ipCurrentMover.MoveCommand.SendToStation(Destination := ipNextStation);
					IF CommandResult.Busy THEN
						_MoverQueue.Dequeue();
						StationState := E_XplanarStationState.CycleComplete;
					END_IF
				END_IF
			END_IF

		E_XPlanarStationState.SendQueue: //Send the mover queue away
			IF i <= _NumMoversRequired THEN
				IF _MoverQueue.Queue[1].Destination <> 0 AND _MoverQueue.Queue[1].Destination.ID <> _ID THEN
					CommandResult := MoverQueue.Queue[1].MoveCommand.SendToStation(Destination := _MoverQueue.Queue[1].Destination);
					IF CommandResult.Busy THEN
						_MoverQueue.Dequeue();
						i := i + 1;
					END_IF
				ELSE
					CommandResult := MoverQueue.Queue[1].MoveCommand.SendToStation(Destination := ipNextStation);
					IF CommandResult.Busy THEN
						_MoverQueue.Dequeue();
						i := i + 1;
					END_IF
				END_IF
			ELSE
				i			 := 1;
				StationState := E_XplanarStationState.CycleComplete;
			END_IF

		E_XplanarStationState.CycleComplete: //Mover on its way out
			_StationReady := FALSE;
			StationState  := E_XplanarStationState.StationIdle;
			
		E_XPlanarStationState.StationError:
			_Error := TRUE;
			
	END_CASE
ELSE
	_StationComplete := FALSE;
	_StationReady	 := FALSE;
	StationState	 := E_XplanarStationState.StationIdle;
END_IF
END_METHOD

PROPERTY HasMover : BOOL
GET
HasMover := _HasMover;
END_GET
SET
_HasMover := HasMover;
END_SET
END_PROPERTY

PROPERTY ID : UDINT
GET
ID := _ID;
END_GET
SET
_ID := ID;
END_SET
END_PROPERTY

PROPERTY MoverDetected : BOOL
GET
END_GET
END_PROPERTY

PROPERTY MoverQueue : REFERENCE TO FB_MoverQueue
GET
MoverQueue ref= _MoverQueue;
END_GET
END_PROPERTY

PROPERTY NextStation : I_XPlanarStation
GET
NextStation := ipNextStation;
END_GET
SET
ipNextStation := NextStation;
END_SET
END_PROPERTY

PROPERTY NumMoversRequired : UDINT
GET
NumMoversRequired := _NumMoversRequired;
END_GET
SET
_NumMoversRequired := NumMoversRequired;
END_SET
END_PROPERTY

PROPERTY Position : REFERENCE TO PositionXYC
GET
Position ref= _Position;
END_GET
END_PROPERTY

METHOD Reset : BOOL
StationState := E_XplanarStationState.StationIdle;
PrepState	 := 0;
_Error		 := FALSE;
Reset		 := true;
END_METHOD

PROPERTY Size : REFERENCE TO Position2D_LREAL
GET
Size ref= _Size;
END_GET
END_PROPERTY

PROPERTY StationComplete : BOOL
SET
_StationComplete := StationComplete;
END_SET
END_PROPERTY

PROPERTY StationReady : BOOL
GET
StationReady := _StationReady;
END_GET
END_PROPERTY

PROPERTY StationType : E_StationType
GET
StationType := _StationType;
END_GET
SET
_StationType := StationType;
END_SET
END_PROPERTY

PROPERTY TrackID : UDINT
GET
TrackID := ipTrackID;
END_GET
SET
ipTrackID := TrackID;
END_SET
END_PROPERTY

METHOD CyclicLogic
IF _ID > 0 AND _ID <= SystemParameters.STATION_COUNT THEN
	XPlanarHMI.StationObjects[_ID].Width  := TO_DINT(_Size.x);
	XPlanarHMI.StationObjects[_ID].Height := TO_DINT(_Size.y);
	XPlanarHMI.StationObjects[_ID].X	   := TO_DINT(_Position.x);
	XPlanarHMI.StationObjects[_ID].Y	   := TO_DINT(_Position.y);
END_IF

SUPER^.CyclicLogic();
END_METHOD

PROPERTY Name : STRING
GET
Name := _Name;
END_GET
SET
_Name := Name;
END_SET
END_PROPERTY

METHOD WatchForMover
VAR_INST
	idx : UDINT;
END_VAR
FOR idx := 1 TO SystemParameters.MOVER_COUNT DO
	IF ip.Movers[idx] <> 0 THEN
		IF _Position.x > 0 AND _Position.y > 0 THEN
			IF (ip.Movers[idx].ActualPosition.x + SystemParameters.AssumedMoverSize >= _Position.x - (_Size.x / 2) AND ip.Movers[idx].ActualPosition.x - SystemParameters.AssumedMoverSize <= _Position.x + (_Size.x / 2)) AND
			   (ip.Movers[idx].ActualPosition.y + SystemParameters.AssumedMoverSize >= _Position.y - (_Size.y / 2) AND ip.Movers[idx].ActualPosition.y - SystemParameters.AssumedMoverSize <= _Position.y + (_Size.y / 2)) THEN
				IF ip.Movers[idx].Destination <> 0 THEN
					IF ip.Movers[idx].Destination.ID = _ID AND NOT ip.Movers[idx].InStation THEN
						_MoverQueue.Enqueue(ip.Movers[idx]);
						IF SystemParameters.EnableCommandTracing THEN
							Trace(CONCAT(CONCAT('Mover ', TO_STRING(ip.Movers[idx].MoverIndex)), CONCAT(' Queued in station ', TO_STRING(_ID))));
						END_IF
					END_IF
				END_IF
			END_IF
		END_IF
	END_IF
END_FOR

IF _MoverQueue.Count > 0 THEN
	_HasMover	   := TRUE;
	ipCurrentMover := _MoverQueue.FirstMover;
ELSE
	_HasMover	   := FALSE;
	ipCurrentMover := 0;
END_IF

IF _HasMover AND ipCurrentMover <> 0 THEN
	IF ipCurrentMover <> 0 THEN
		CASE _StationType OF
			E_StationType.Process:
				_StationReady := NOT ipCurrentMover.Status.Busy.busyMover;

			E_StationType.MultiMover:
				_StationReady := NOT ipCurrentMover.Status.Busy.busyMover AND (_MoverQueue.Count = _NumMoversRequired);

			E_StationType.DecisionPoint:
				_StationReady := _HasMover;
		END_CASE
	END_IF
END_IF
END_METHOD

END_FUNCTION_BLOCK

// Tile/FB_XPlanarTile
FUNCTION_BLOCK FB_XPlanarTile EXTENDS FB_CyclicFB
VAR
	ipTileTcIo			: I_TcIoXPlanarTile;
	_Index				: UINT;
	_Part				: UINT := 1;
	_Btn				: STRING(13);
	_DcLinkVoltage		: UINT;
	_DcLinkOk			: BOOL;
	_TimeToShutdown		: UDINT;
	_ObservedPower		: LREAL;
	_OverLimitFactor	: LREAL;
	_DiagData			: POINTER TO ST_CoeDriveDiagData;
	_Position			: ST_TcIoTilePositionOnPart;
	_Temperatures		: ST_TileTemperatures;
	CoEUpdateTimer		: TON;
	CriticalUpdateTimer : TON;
	DiagDataResult		: ULINT;
END_VAR

PROPERTY Btn : STRING(13)
GET
Btn := _Btn;
END_GET
END_PROPERTY

METHOD PUBLIC CyclicLogic
VAR_INST
	Update : BOOL;
	test   : DINT;
END_VAR
IF XPlanar.OperationMode = Tc3_XPlanarUtility.OperationMode.Normal THEN
	IF SystemParameters.TileDiagUpdate > 0 THEN
		CoEUpdateTimer(IN := NOT Update, PT := TO_TIME(SystemParameters.TileDiagUpdate) * 1000);
		IF CoEUpdateTimer.Q THEN
			Update := TRUE;
		END_IF

		test := SIZEOF(_diagdata);

		//Update the tile diagnostic data
		IF update AND_THEN XPlanar.EnvironmentTcIo.XpuTcIo(1).TileTcIo(_Part, Index).CoE.DiagData.Update() THEN
			_DiagData := XPlanar.EnvironmentTcIo.XpuTcIo(1).TileTcIo(_Part, Index).CoE.DiagData.All;
			_DcLinkOk := XPlanar.EnvironmentTcIo.XpuTcIo(1).TileTcIo(_Part, Index).CoE.DiagData.DcLinkOk;
			Update	  := FALSE;
		END_IF

		CriticalUpdateTimer(IN := NOT CriticalUpdateTimer.Q, PT := T#1S);
		IF CriticalUpdateTimer.Q THEN
			_TimeToShutdown	 := XPlanar.EnvironmentTcIo.XpuTcIo(1).TileTcIo(_Part, Index).GetCoeTimeToShutdown();
			_ObservedPower	 := XPlanar.EnvironmentTcIo.XpuTcIo(1).TileTcIo(_Part, Index).GetObservedTilePower();
			_OverLimitFactor := XPlanar.EnvironmentTcIo.XpuTcIo(1).TileTcIo(_Part, Index).GetPowerOverLimitFactor();
		END_IF
	ELSE
		Update := FALSE;
	END_IF
END_IF
END_METHOD

PROPERTY DcLinkOk : BOOL
GET
DcLinkOk := _DcLinkOk;
END_GET
END_PROPERTY

PROPERTY Index : UINT
GET
Index := _Index;
END_GET
SET
_Index := Index;
END_SET
END_PROPERTY

METHOD Initialize : BOOL
//Get BTN of tile
_Btn := XPlanar.EnvironmentTcIo.XpuTcIo(1).TileTcIo(_Part, _Index).GetBtn();

//Get the configured position of the tile
_Position := XPlanar.EnvironmentTcIo.XpuTcIo(1).TileTcIo(_Part, _Index).TilePositionOnPart();

//Update the object array for HMI
XPlanarHMI.TileObjects[_Index].X	   := _Position.X;
XPlanarHMI.TileObjects[_Index].Width  := 240; //Currently the only size, but will change in the future.
XPlanarHMI.TileObjects[_Index].Y	   := _Position.Y;
XPlanarHMI.TileObjects[_Index].Height := 240; //Currently the only size, but will change in the future.

//Get initial diagnostic data
IF _Part > 0 AND _Index > 0 THEN
	ipTileTcIo := XPlanar.EnvironmentTcIo.XpuTcIo(1).TileTcIo(_Part, Index);
	IF XPlanar.OperationMode = Tc3_XPlanarUtility.OperationMode.Normal THEN
		IF XPlanar.EnvironmentTcIo.XpuTcIo(1).TileTcIo(_Part, _Index).CoE.DiagData.Update() THEN
			_DiagData  := XPlanar.EnvironmentTcIo.XpuTcIo(1).TileTcIo(_Part, _Index).CoE.DiagData.All;
			Initialize := TRUE;
		END_IF
	END_IF
END_IF
END_METHOD

PROPERTY PartIndex : UINT
GET
PartIndex := _Part;
END_GET
SET
_Part := PartIndex;
END_SET
END_PROPERTY

PROPERTY PositionOnPart : REFERENCE TO ST_TcIoTilePositionOnPart
GET
PositionOnPart ref= _Position;
END_GET
END_PROPERTY

PROPERTY Temperatures : REFERENCE TO ST_TileTemperatures
GET
Temperatures ref= _Temperatures;
END_GET
END_PROPERTY

PROPERTY TimeToShutdown : UDINT
GET
TimeToShutdown := _TimeToShutdown;
END_GET
END_PROPERTY

METHOD Update
VAR_INPUT
END_VAR
XPlanar.EnvironmentTcIo.XpuTcIo(1).TileTcIo(_Part, Index).CoE.DiagData.Update();
_DiagData		 := XPlanar.EnvironmentTcIo.XpuTcIo(1).TileTcIo(_Part, Index).CoE.DiagData.All;
_DcLinkOk		 := XPlanar.EnvironmentTcIo.XpuTcIo(1).TileTcIo(_Part, Index).CoE.DiagData.DcLinkOk;
_TimeToShutdown	 := XPlanar.EnvironmentTcIo.XpuTcIo(1).TileTcIo(_Part, Index).GetCoeTimeToShutdown();
_ObservedPower	 := XPlanar.EnvironmentTcIo.XpuTcIo(1).TileTcIo(_Part, Index).GetObservedTilePower();
_OverLimitFactor := XPlanar.EnvironmentTcIo.XpuTcIo(1).TileTcIo(_Part, Index).GetPowerOverLimitFactor();
END_METHOD

PROPERTY Utility : I_TcIoXPlanarTile
GET
IF ipTileTcIo <> 0 THEN
	Utility := ipTileTcIo;
end_if
END_GET
END_PROPERTY

END_FUNCTION_BLOCK

// Tile/I_XPlanarTile
INTERFACE I_XPlanarTile EXTENDS I_BaseFB

PROPERTY Btn : STRING(13)
GET
END_GET
END_PROPERTY

PROPERTY DcLinkOk : BOOL
GET
END_GET
END_PROPERTY

PROPERTY Index : UINT
GET
END_GET
SET
END_SET
END_PROPERTY

PROPERTY PartIndex : UINT
GET
END_GET
SET
END_SET
END_PROPERTY

PROPERTY PositionOnPart : REFERENCE TO ST_TcIoTilePositionOnPart
GET
END_GET
END_PROPERTY

PROPERTY Temperatures : REFERENCE TO ST_TileTemperatures
GET
END_GET
END_PROPERTY

PROPERTY TimeToShutdown : UDINT
GET
END_GET
END_PROPERTY

METHOD Update
VAR_INPUT
END_VAR
END_METHOD

PROPERTY Utility : I_TcIoXPlanarTile
GET
END_GET
END_PROPERTY

END_INTERFACE

// Track/TaskClasses/FB_AddTrackToGroup
FUNCTION_BLOCK FB_AddTrackToGroup EXTENDS FB_TrackTaskResult
VAR
END_VAR

METHOD Execute : I_PlanarTaskResult
VAR_INPUT
	refGroup : REFERENCE TO MC_PlanarGroup;
END_VAR
_Done	 := FALSE;
_Error	 := FALSE;
_Busy	 := FALSE;
_ErrorID := 0;
ipTrack.pm.AddToGroup(_PlanarFb, refGroup);
Execute := THIS^;

//Heartbeat that the method is active
ExecuteWatchdog := ExecuteWatchdog + 1;
END_METHOD

END_FUNCTION_BLOCK

// XPlanarResultClasses/FB_TrackTaskResult
FUNCTION_BLOCK FB_TrackTaskResult EXTENDS FB_PlanarFeedbackResult
VAR
	ipTrack	   : I_XPlanarTrack;
END_VAR

PROPERTY Track : I_XplanarTrack
SET
ipTrack := Track;
END_SET
END_PROPERTY

END_FUNCTION_BLOCK

// Track/TaskClasses/FB_AppendLine
FUNCTION_BLOCK FB_AppendLine EXTENDS FB_TrackTaskResult
VAR
	StartPoint : PositionXYC;
	EndPoint   : PositionXYC;
END_VAR

METHOD Execute : I_PlanarTaskResult
VAR_INPUT
	StartPointX : LREAL;
	StartPointY : LREAL;
	EndPointX	: LREAL;
	EndPointY	: LREAL;
END_VAR
IF NOT HasRun THEN
	_Done	 := FALSE;
	_Error	 := FALSE;
	_Busy	 := FALSE;
	_ErrorID := 0;
	StartPoint.SetValuesXY(StartPointX, StartPointY);
	EndPoint.SetValuesXY(EndPointX, EndPointY);
	ipTrack.pm.AppendLine(_PlanarFb, StartPoint, EndPoint);
	HasRun := TRUE;
END_IF

Execute := THIS^;

//Heartbeat that the method is active
ExecuteWatchdog := ExecuteWatchdog + 1;
END_METHOD

END_FUNCTION_BLOCK

// Track/TaskClasses/FB_AppendPoint
FUNCTION_BLOCK FB_AppendPoint EXTENDS FB_TrackTaskResult
VAR
	Position : PositionXYC;
END_VAR

METHOD Execute : I_PlanarTaskResult
VAR_INPUT
	XPoint : LREAL;
	YPoint : LREAL;
END_VAR
IF NOT HasRun THEN
	_Done	 := FALSE;
	_Error	 := FALSE;
	_Busy	 := FALSE;
	_ErrorID := 0;
	Position.SetValuesXY(XPoint, YPoint);
	ipTrack.pm.AppendPosition(_PlanarFb, Position);
	HasRun := TRUE;
END_IF

Execute := THIS^;

//Heartbeat that the method is active
ExecuteWatchdog := ExecuteWatchdog + 1;
END_METHOD

END_FUNCTION_BLOCK

// Track/TaskClasses/FB_BuildTrack
FUNCTION_BLOCK FB_BuildTrack EXTENDS FB_TrackTaskResult
VAR
	BuildTrack	: BOOL;
END_VAR

METHOD Execute : I_PlanarTaskResult
IF NOT HasRun THEN
	_Done	   := FALSE;
	_Error	   := FALSE;
	_Busy	   := FALSE;
	_ErrorID   := 0;
	BuildTrack := TRUE;
	HasRun	   := TRUE;
END_IF

Execute := THIS^;

//Heartbeat that the method is active
ExecuteWatchdog := ExecuteWatchdog + 1;
END_METHOD

METHOD PUBLIC Update
VAR_INST
	WatchdogCheck : UDINT;
	i			  : UDINT := 1;
END_VAR
_PlanarFb.Update();
CASE TaskState OF
	0: //Init
		THIS^._Busy := FALSE;
		IF BuildTrack THEN
			THIS^._Done	   := FALSE;
			THIS^._Error   := FALSE;
			THIS^._ErrorID := 0;
			THIS^._Busy	   := TRUE;
			BuildTrack	   := FALSE;
			i			   := 1;
			TaskState	   := TaskState + 10;
		END_IF

	10: //Set StartFromTrack
		IF ipTrack.Definition.StartFromTrackID > 0 THEN
			ipTrack.pm.StartFromTrack(_PlanarFb, ip.Tracks[ipTrack.Definition.StartFromTrackID].pm);
			TaskState := TaskState + 1;
		ELSE
			TaskState := TaskState + 10;
		END_IF

	11: //Watch Command Feedback
		IF _PlanarFb.Done THEN
			TaskState := 20;
		ELSIF _PlanarFb.Error THEN
			THIS^._Error			  := TRUE;
			THIS^._ErrorID			  := _PlanarFb.ErrorId;
			THIS^._BlockingObjectInfo := _PlanarFb.objectInfo;
			TaskState				  := 0;
		END_IF

	20: //Append Track Objects
		IF ipTrack.Definition.Items[i].StartPoint.x > 0 THEN
			CASE ipTrack.Definition.Items[i].ItemType OF
				Point:
					ipTrack.pm.AppendPosition(_PlanarFb, ipTrack.Definition.Items[i].StartPoint);

				Line:
					IF ipTrack.Definition.Items[i].EndPoint.x > 0 THEN
						ipTrack.pm.AppendLine(_PlanarFb, ipTrack.Definition.Items[i].StartPoint, ipTrack.Definition.Items[i].EndPoint);
					ELSE
						THIS^._Error			  := TRUE;
						THIS^._ErrorID			  := 9999;
						TaskState				  := 0;	
					END_IF					
					
				Circle:
					ipTrack.pm.AppendCircle(_PlanarFb,
									   ipTrack.Definition.Items[i].StartPoint,
									   ipTrack.Definition.Items[i].EndPoint,
									   ipTrack.Definition.Items[i].CenterPoint,
									   ipTrack.Definition.Items[i].CircleClockwise);
			END_CASE

			TaskState := TaskState + 1;
		ELSE
			TaskState := TaskState + 10; //No Object Defined Exit the loop
		END_IF

	21: //Watch Command Feedback
		IF _PlanarFb.Done THEN
			IF i < SystemParameters.MAX_OBJECTS_PER_TRACK THEN
				i		  := i + 1;
				TaskState := 20;
			ELSE
				i		  := 1;
				TaskState := 30;
			END_IF
		ELSIF _PlanarFb.Error THEN
			THIS^._Error			  := TRUE;
			THIS^._ErrorID			  := _PlanarFb.ErrorId;
			THIS^._BlockingObjectInfo := _PlanarFb.objectInfo;
			TaskState				  := 0;
		END_IF

	30: //Set EndAtTrack
		IF ipTrack.Definition.EndAtTrackID > 0 THEN
			ipTrack.pm.EndAtTrack(_PlanarFb, ip.Tracks[ipTrack.Definition.EndAtTrackID].pm);
			TaskState := TaskState + 1;
		ELSIF ipTrack.Definition.CloseLoop THEN
			ipTrack.pm.CloseLoop(_PlanarFb);
			TaskState := TaskState + 1;
		ELSE
			TaskState := TaskState + 10;
		END_IF

	31: //Watch Command Feedback
		IF _PlanarFb.Done THEN
			TaskState := 40;
		ELSIF _PlanarFb.Error THEN
			THIS^._Error			  := TRUE;
			THIS^._ErrorID			  := _PlanarFb.ErrorId;
			THIS^._BlockingObjectInfo := _PlanarFb.objectInfo;
			TaskState				  := 0;
		END_IF

	40: //Build Complete
		THIS^._Done := TRUE;
		TaskState	:= 0;
END_CASE

IF ExecuteWatchdog <> WatchdogCheck THEN
	WatchdogCheck := ExecuteWatchdog;
ELSE
	HasRun			:= FALSE;
	ExecuteWatchdog := 0;
END_IF
END_METHOD

END_FUNCTION_BLOCK

// Track/TaskClasses/FB_ClearSegment
FUNCTION_BLOCK FB_ClearSegment EXTENDS FB_TrackTaskResult
VAR
END_VAR

METHOD Execute : I_PlanarTaskResult
IF NOT HasRun THEN
	_Done	 := FALSE;
	_Error	 := FALSE;
	_Busy	 := FALSE;
	_ErrorID := 0;
	ipTrack.pm.Clear(_PlanarFb);
	HasRun := TRUE;
END_IF

Execute := THIS^;

//Heartbeat that the method is active
ExecuteWatchdog := ExecuteWatchdog + 1;
END_METHOD

END_FUNCTION_BLOCK

// Track/TaskClasses/FB_CloseLoop
FUNCTION_BLOCK FB_CloseLoop EXTENDS FB_TrackTaskResult
VAR
END_VAR

METHOD Execute : I_PlanarTaskResult
IF NOT HasRun THEN
	_Done	 := FALSE;
	_Error	 := FALSE;
	_Busy	 := FALSE;
	_ErrorID := 0;
	ipTrack.pm.CloseLoop(_PlanarFb);
	HasRun := TRUE;
END_IF

Execute := THIS^;

//Heartbeat that the method is active
ExecuteWatchdog := ExecuteWatchdog + 1;
END_METHOD

END_FUNCTION_BLOCK

// Track/TaskClasses/FB_DisableTrack
FUNCTION_BLOCK FB_DisableTrack EXTENDS FB_TrackTaskResult
VAR
END_VAR

METHOD Execute : I_PlanarTaskResult
VAR_INPUT
END_VAR
IF ipTrack.Status.State = Mc_Planar_State.Enabled THEN
	_Done	 := FALSE;
	_Error	 := FALSE;
	_Busy	 := FALSE;
	_ErrorID := 0;
	ipTrack.pm.Disable(_PlanarFb);
END_IF

Execute := THIS^;

//Heartbeat that the method is active
ExecuteWatchdog := ExecuteWatchdog + 1;
END_METHOD

END_FUNCTION_BLOCK

// Track/TaskClasses/FB_EnableTrack
FUNCTION_BLOCK FB_EnableTrack EXTENDS FB_TrackTaskResult
VAR
END_VAR

METHOD Execute : I_PlanarTaskResult
VAR_INPUT
END_VAR
IF ipTrack.Status.State = Mc_Planar_State.Disabled THEN
	_Done	 := FALSE;
	_Error	 := FALSE;
	_Busy	 := FALSE;
	_ErrorID := 0;
	ipTrack.pm.Enable(_PlanarFb);
END_IF

Execute := THIS^;

//Heartbeat that the method is active
ExecuteWatchdog := ExecuteWatchdog + 1;
END_METHOD

END_FUNCTION_BLOCK

// Track/TaskClasses/FB_SetEndAtTrack
FUNCTION_BLOCK FB_SetEndAtTrack EXTENDS FB_TrackTaskResult
VAR
	Options : ST_EndAtTrackAdvancedOptions;
END_VAR

METHOD Execute : I_PlanarTaskResult
VAR_INPUT
	SegmentID : UDINT;
END_VAR
IF NOT HasRun AND (SegmentID > 0 AND SegmentID <= SystemParameters.TRACK_COUNT) THEN
	_Done	 := FALSE;
	_Error	 := FALSE;
	_Busy	 := FALSE;
	_ErrorID := 0;
	ipTrack.pm.EndAtTrack(_PlanarFb, ip.Tracks[SegmentID].pm);
	HasRun := TRUE;
END_IF

Execute := THIS^;

//Heartbeat that the method is active
ExecuteWatchdog := ExecuteWatchdog + 1;
END_METHOD

END_FUNCTION_BLOCK

// Track/TaskClasses/FB_SetStartFromTrack
FUNCTION_BLOCK FB_SetStartFromTrack EXTENDS FB_TrackTaskResult
VAR
	Options : ST_StartFromTrackAdvancedOptions;
END_VAR

METHOD Execute : I_PlanarTaskResult
VAR_INPUT
	SegmentID : UDINT;
END_VAR
IF NOT HasRun AND (SegmentID > 0 AND SegmentID <= SystemParameters.TRACK_COUNT) THEN
	_Done	 := FALSE;
	_Error	 := FALSE;
	_Busy	 := FALSE;
	_ErrorID := 0;
	ipTrack.pm.StartFromTrack(_PlanarFb, ip.Tracks[SegmentID].pm);
	HasRun := TRUE;
END_IF

Execute := THIS^;

//Heartbeat that the method is active
ExecuteWatchdog := ExecuteWatchdog + 1;
END_METHOD

END_FUNCTION_BLOCK

// Track/TaskClasses/FB_TrackReset
FUNCTION_BLOCK FB_TrackReset EXTENDS FB_TrackTaskResult
VAR
END_VAR

METHOD Execute : I_PlanarTaskResult
IF NOT HasRun THEN
	_Done	 := FALSE;
	_Error	 := FALSE;
	_Busy	 := FALSE;
	_ErrorID := 0;
	ipTrack.pm.Reset(_PlanarFb);
	HasRun := TRUE;
END_IF

Execute := THIS^;

//Heartbeat that the method is active
ExecuteWatchdog := ExecuteWatchdog + 1;
END_METHOD

END_FUNCTION_BLOCK

// Track/FB_XPlanarTrackSegment
FUNCTION_BLOCK FB_XPlanarTrackSegment EXTENDS FB_CyclicFB IMPLEMENTS I_XPlanarTrack
VAR
	//Planar Track 
	_Track			: MC_PlanarTrack;
	_Definition		: ST_TrackDefinition;
	ipMcPlanarTrack : I_McPlanarTrack;

	//Track Segment Task Classes
	AppendLineToSegment	  : FB_AppendLine		 := (Track := THIS^);
	AppendPointToSegment  : FB_AppendPoint		 := (Track := THIS^);
	CloseTheLoop		  : FB_CloseLoop		 := (Track := THIS^);
	EnableTrack			  : FB_EnableTrack		 := (Track := THIS^);
	DisableTrack		  : FB_DisableTrack		 := (Track := THIS^);
	ClearTrackPoints	  : FB_ClearSegment		 := (Track := THIS^);
	AddTrackToGroup		  : FB_AddTrackToGroup	 := (Track := THIS^);
	SetStartFromTrackTask : FB_SetStartFromTrack := (Track := THIS^);
	SetEndAtTrackTask	  : FB_SetEndAtTrack	 := (Track := THIS^);
	ResetTrack			  : FB_TrackReset		 := (Track := THIS^);
	BuildTrack			  : FB_BuildTrack		 := (Track := THIS^);

	//Internal Vars
	_std		 : CDT_MCTOPLC_PLANAR_TRACK;
	_TrackLength : LREAL;
	_TrackID	 : UDINT;
END_VAR

METHOD AddToGroup : I_PlanarTaskResult
VAR_INPUT
	PlanarGroup : REFERENCE TO MC_PlanarGroup;
END_VAR
AddToGroup := AddTrackToGroup.Execute(PlanarGroup);
END_METHOD

METHOD AppendLine : I_PlanarTaskResult
VAR_INPUT
	StartPointX : LREAL;
	StartPointY : LREAL;
	EndPointX	: LREAL;
	EndPointY	: LREAL;
END_VAR

VAR_INST
END_VAR
AppendLine := AppendLineToSegment.Execute(StartPointX,
										  StartPointY,
										  EndPointX,
										  EndPointY);
END_METHOD

METHOD AppendPoint : I_PlanarTaskResult
VAR_INPUT
	XPoint : LREAL;
	YPoint : LREAL;
END_VAR

VAR_INST
END_VAR
AppendPoint := AppendPointToSegment.Execute(XPoint, YPoint);
END_METHOD

METHOD Build : I_PlanarTaskResult
Build := BuildTrack.Execute();
END_METHOD

METHOD Clear : I_PlanarTaskResult
VAR_INST
	nStateReset : UINT;
END_VAR
Clear := ClearTrackPoints.Execute();
END_METHOD

METHOD CloseLoop : I_PlanarTaskResult
CloseLoop := CloseTheLoop.Execute();
END_METHOD

PROPERTY Definition : REFERENCE TO ST_TrackDefinition
GET
Definition ref= _Definition;
END_GET
END_PROPERTY

METHOD Disable : I_PlanarTaskResult
Disable := DisableTrack.Execute();
END_METHOD

{attribute 'TcRpcEnable'}
METHOD Enable : I_PlanarTaskResult
Enable := EnableTrack.Execute();
END_METHOD

METHOD GetTrackPositionAt : LREAL;
VAR_IN_OUT
	Position : PositionXYC;
END_VAR
GetTrackPositionAt := _Track.GetArcLengthClosestTo(Position);
END_METHOD

PROPERTY Index : UDINT
GET
Index := _TrackID;
END_GET
SET
_TrackID := Index;
END_SET
END_PROPERTY

PROPERTY MoverCount : UDINT
GET
MoverCount := _Track.MCTOPLC_STD.MoverCountOnTrack;
END_GET
END_PROPERTY

PROPERTY MovingMoverCount : UDINT
GET
MovingMoverCount := _Track.MCTOPLC_STD.MovingMoverCount;
END_GET
END_PROPERTY

PROPERTY pm : REFERENCE TO MC_PlanarTrack
GET
pm ref= _Track;
END_GET
END_PROPERTY

METHOD Reset : I_PlanarTaskResult
VAR_INPUT
END_VAR
Reset := ResetTrack.Execute();
END_METHOD

METHOD SetEndAtTrack : I_PlanarTaskResult
VAR_INPUT
	SegmentID : UDINT;
END_VAR
SetEndAtTrack := SetEndAtTrackTask.Execute(SegmentID);
END_METHOD

METHOD SetStartFromTrack : I_PlanarTaskResult
VAR_INPUT
	SegmentID : UDINT;
END_VAR
SetStartFromTrack := SetStartFromTrackTask.Execute(SegmentID);
END_METHOD

PROPERTY Status : REFERENCE TO CDT_MCTOPLC_PLANAR_TRACK
GET
Status ref= _std;
END_GET
END_PROPERTY

PROPERTY TrackLength : LREAL
GET
TrackLength := _Track.GetLength();
END_GET
END_PROPERTY

PROPERTY Utility : I_McPlanarTrack
GET
IF ipMcPlanarTrack <> 0 THEN
	Utility := ipMcPlanarTrack;
END_IF
END_GET
SET
ipMcPlanarTrack := Utility;
END_SET
END_PROPERTY

METHOD CyclicLogic
VAR
	Result : BOOL;
END_VAR
_std := _Track.MCTOPLC_STD;
EnableTrack.Update();
DisableTrack.Update();
AppendLineToSegment.Update();
AppendPointToSegment.Update();
ClearTrackPoints.Update();
CloseTheLoop.Update();
AddTrackToGroup.Update();
SetStartFromTrackTask.Update();
SetEndAtTrackTask.Update();
ResetTrack.Update();
BuildTrack.Update();
END_METHOD

END_FUNCTION_BLOCK

// XPlanarComponent/TaskClasses/FB_EnableGroup
FUNCTION_BLOCK FB_EnableGroup EXTENDS FB_PlanarFeedbackResult
VAR
END_VAR

METHOD Execute : I_PlanarTaskResult
IF NOT HasRun AND XPlanar.Group.MCTOPLC_STD.State = MC_PLANAR_STATE.Disabled THEN
	_Done	 := FALSE;
	_Error	 := FALSE;
	_Busy	 := FALSE;
	_ErrorID := 0;
	XPlanar.Group.Enable(_PlanarFb);
	HasRun := TRUE;
END_IF

Execute := THIS^;

//Heartbeat that the method is active
ExecuteWatchdog := ExecuteWatchdog + 1;
END_METHOD

END_FUNCTION_BLOCK

// XPlanarComponent/TaskClasses/FB_MoverIdentification
FUNCTION_BLOCK FB_MoverIdentification EXTENDS FB_PlanarFeedbackResult
VAR
	_MoverIdentificationStatus : CoordinatedMoverCommStatus;
	_CoordinatedMoverComm	   : CoordinatedMoverCommCommand;
END_VAR

METHOD Execute : I_PlanarTaskResult
IF XPlanar.OperationMode = XPlanarOperationMode.Normal THEN
	IF NOT HasRun THEN
		_Done	 := FALSE;
		_Error	 := FALSE;
		_Busy	 := FALSE;
		_ErrorID := 0;
		Xplanar.EnvironmentTcIo.XpuTcIo(1).SetCoordMoverCommunicationCmd(_CoordinatedMoverComm);
		HasRun := TRUE;
	END_IF
END_IF

Execute := THIS^;

//Heartbeat that the method is active
ExecuteWatchdog := ExecuteWatchdog + 1;
END_METHOD

METHOD Update
VAR_INST
	WatchdogCheck : UDINT;
END_VAR
IF ExecuteWatchdog <> WatchdogCheck THEN
	_MoverIdentificationStatus := XPlanar.EnvironmentTcIo.XpuTcIo(1).GetCoordMoverCommStatus();
	WatchdogCheck			   := ExecuteWatchdog;
ELSE
	HasRun := FALSE;
	ExecuteWatchdog := 0;
END_IF

THIS^.Busy	:= _MoverIdentificationStatus = CoordinatedMoverCommStatus.CommunicationInProcess;
THIS^.Done	:= _MoverIdentificationStatus = CoordinatedMoverCommStatus.CommunicationSuccessful;
THIS^.Error := _MoverIdentificationStatus = CoordinatedMoverCommStatus.CommunicationFailed;
END_METHOD

END_FUNCTION_BLOCK

// XPlanarComponent/TaskClasses/FB_MoverRedetection
FUNCTION_BLOCK FB_MoverRedetection EXTENDS FB_PlanarFeedbackResult
VAR
	_MoverDetectionStatus : MoverDetectionStatus;
	_MoverDetectionInfo	  : ST_TcIoMoverDetectionInfos;
END_VAR

METHOD Execute : I_PlanarTaskResult
IF NOT HasRun THEN
	_Done	 := FALSE;
	_Error	 := FALSE;
	_Busy	 := FALSE;
	_ErrorID := 0;
	Xplanar.EnvironmentTcIo.XpuTcIo(1).SetStartMoverRedetection();
	HasRun := TRUE;
END_IF

IF _Done THEN
	_MoverDetectionInfo := XPlanar.EnvironmentTcIo.XpuTcIo(1).GetMoverDetectionInfos();
END_IF

Execute := THIS^;

//Heartbeat that the method is active
ExecuteWatchdog := ExecuteWatchdog + 1;
END_METHOD

METHOD Update
VAR_INST
	WatchdogCheck : UDINT;
END_VAR
IF ExecuteWatchdog <> WatchdogCheck THEN
	_MoverDetectionStatus := XPlanar.EnvironmentTcIo.XpuTcIo(1).GetMoverDetectionStatus();
	WatchdogCheck		  := ExecuteWatchdog;
ELSE
	HasRun := FALSE;
	ExecuteWatchdog := 0;
END_IF

THIS^.Busy	:= _MoverDetectionStatus = MoverDetectionStatus.DetectionInProcess;
THIS^.Done	:= _MoverDetectionStatus = MoverDetectionStatus.DetectionSuccessful;
THIS^.Error := _MoverDetectionStatus = MoverDetectionStatus.NotInitialized;
END_METHOD

END_FUNCTION_BLOCK

// XPlanarComponent/TaskClasses/FB_ResetGroup
FUNCTION_BLOCK FB_ResetGroup EXTENDS FB_PlanarFeedbackResult
VAR
END_VAR

METHOD Execute : I_PlanarTaskResult
IF NOT HasRun AND XPlanar.Group.Error THEN
	_Done	 := FALSE;
	_Error	 := FALSE;
	_Busy	 := FALSE;
	_ErrorID := 0;
	XPlanar.Group.Reset(_PlanarFb);
	HasRun := TRUE;
END_IF

Execute := THIS^;

//Heartbeat that the method is active
ExecuteWatchdog := ExecuteWatchdog + 1;
END_METHOD

END_FUNCTION_BLOCK

// XPlanarComponent/TaskClasses/FB_ResetXPlanar
FUNCTION_BLOCK FB_ResetXPlanar EXTENDS FB_PlanarFeedbackResult
VAR
	_MoverDetectionStatus : MoverDetectionStatus;
	_MoverDetectionInfo	  : ST_TcIoMoverDetectionInfos;
END_VAR

METHOD Execute : I_PlanarTaskResult
VAR_INST
	i	: UDINT;
	MoverResetResult	: I_PlanarTaskResult;
	TrackResetResult	: I_PlanarTaskResult;
END_VAR
CASE TaskState OF
	0: //Init
		i		  := 1;
		_Done	  := FALSE;
		_Error	  := FALSE;
		TaskState := TaskState + 10;

	10: //Reset Movers
		IF i <= SystemParameters.MOVER_COUNT THEN
			MoverResetResult := ip.Movers[i].Reset();
			IF MoverResetResult.Done THEN
				TaskState := TaskState + 1;
			ELSIF MoverResetResult.Error THEN
				TaskState := 997;
			END_IF
		ELSE
			i		  := 1;
			TaskState := TaskState + 10;
		END_IF

	11: //Increment Index
		i		  := i + 1;
		TaskState := TaskState - 1;

	20: //Reset Track Segments
		IF i <= SystemParameters.TRACK_COUNT THEN
			TrackResetResult := ip.Tracks[i].Reset();
			IF TrackResetResult.Done THEN
				TaskState := TaskState + 1;
			ELSIF TrackResetResult.Error THEN
				TaskState := 998;
			END_IF
		ELSE
			i		  := 1;
			TaskState := TaskState + 10;
		END_IF

	21: //Increment Index
		i		  := i + 1;
		TaskState := TaskState - 1;

	30: //Reset Group
		IF XPlanar.Group.Error THEN
			XPlanar.Group.Reset(_PlanarFb);
		END_IF

		TaskState := TaskState + 10;

	40: //Check Group Reset Command Feedback
		IF _PlanarFb.Done OR NOT XPlanar.Group.Error THEN
			TaskState := TaskState + 10;
		ELSIF _PlanarFb.Error THEN
			TaskState := 999;
		END_IF

	50: //Reset Complete
		_Done := TRUE;

	997: //Mover Reset Error
		_Error				:= MoverResetResult.Error;
		_ErrorID			:= MoverResetResult.ErrorID;
		_BlockingObjectInfo := MoverResetResult.BlockingObjectInfo;

	998: //Mover Reset Error
		_Error				:= TrackResetResult.Error;
		_ErrorID			:= TrackResetResult.ErrorID;
		_BlockingObjectInfo := TrackResetResult.BlockingObjectInfo;

	999: //Group Reset Error
		_Error				:= _PlanarFb.Error;
		_ErrorID			:= _PlanarFb.ErrorId;
		_BlockingObjectInfo := _PlanarFb.objectInfo;
END_CASE

Execute := THIS^;

//Heartbeat that the method is active
ExecuteWatchdog := ExecuteWatchdog + 1;
END_METHOD

METHOD Update
VAR_INST
	WatchdogCheck : UDINT;
END_VAR
IF ExecuteWatchdog <> WatchdogCheck THEN
	WatchdogCheck := ExecuteWatchdog;
ELSE
	HasRun			:= FALSE;
	TaskState		:= 0;
	ExecuteWatchdog := 0;
END_IF

_PlanarFb.Update();
THIS^.Busy := TaskState > 0 AND TaskState < 50;
END_METHOD

END_FUNCTION_BLOCK

// XPlanarComponent/FB_Component_XPlanar
FUNCTION_BLOCK FB_Component_XPlanar EXTENDS FB_ComponentBase
VAR
	XPlanarBaseAlarms : ARRAY[1..XPLANAR_BASE_ALARM_COUNT] OF FB_TcAlarm;
	Parts			  : ARRAY[1..Param_TcIoXPlanarEnvironment.MaxParts] OF FB_XPlanarPart;
	Tiles			  : ARRAY[1..Param_TcIoXPlanarEnvironment.MaxTiles] OF FB_XPlanarTile;
	ipMoverCyclic	  : ARRAY[1..SystemParameters.MOVER_COUNT] OF I_CyclicFB;
	ipTrackCyclic	  : ARRAY[1..SystemParameters.TRACK_COUNT] OF I_CyclicFB;
	UtilityVisu		  : FB_XPlanarUtilityVisu;

	//System Level Tasks
	EnablePlanarGroup	: FB_EnableGroup;
	MoverDetection		: FB_MoverRedetection;
	MoverIdentification : FB_MoverIdentification;
	XPlanarReset		: FB_ResetXPlanar;

	//Helper Vars
	_OperationMode		: XPlanarOperationMode;
	_Xpu				: I_TcIoXPlanarProcessingUnit;
	_TracksInitialized	: BOOL;
	_MoverDetectionInfo : ST_TcIoMoverDetectionInfos;
	AbortState			: UDINT;
END_VAR

VAR CONSTANT
	XPLANAR_BASE_ALARM_COUNT : UINT := 6; // Number of defined events configured in the tmc file
END_VAR

//! @summary Initializes event function blocks using this components's name
{attribute 'call_after_online_change_slot' := '<slot>'}
METHOD PROTECTED CreateEvents

//! @description This method is called by <c>Initialize()</c> as required
F_CreateAllEventsInClass(Alarms		:= XPlanarBaseAlarms,
						 ClassSize	:= SIZEOF(TC_EVENTS.XPlanarApplicationEventClass),
						 pInitEvent := ADR(TC_EVENTS.XPlanarApplicationEventClass.InitReferenceEvent),
						 Prefix		:= Name);

SUPER^.CreateEvents();
END_METHOD

//! Provides basic error detection and event handling for this component
METHOD PROTECTED Monitoring
(*! @descriptionThis method is called cyclically by <c>CyclicLogic()</c>*)
VAR
	i	   : UDINT;
	Result : HRESULT;
END_VAR
SUPER^.Monitoring();
FOR i := 1 TO SystemParameters.MOVER_COUNT DO
	IF ip.Movers[i] <> 0 THEN
		IF ip.Movers[i].Status.State = MC_PLANAR_STATE.Error AND NOT XPlanarBaseAlarms[E_XPlanarApplicationEventClass.MoverError].bRaised THEN
			RaiseAlarmWithStrings(Alarm := XPlanarBaseAlarms[E_XPlanarApplicationEventClass.MoverError], CONCAT('Mover ', ip.Movers[i].MoverBTN), 'Faulted');
		END_IF

		IF ip.Movers[i].Error AND NOT XPlanarBaseAlarms[E_XPlanarApplicationEventClass.CommandError].bRaised THEN
			RaiseEventWithStrings(Alarm := XPlanarBaseAlarms[E_XPlanarApplicationEventClass.CommandError], CONCAT('Mover ', TO_STRING(ip.Movers[i].MoverIndex)), TO_STRING(ip.Movers[i].ErrorID));
		END_IF
	END_IF
END_FOR

//Catch the XPlanar errors
_CurrentAlarmSeverity := F_GetMaxSeverityRaised(Alarms := XPlanarBaseAlarms, CurrentSeverity := _CurrentAlarmSeverity);
END_METHOD

//! @summary This method serves as the entry point for all underlying FB logic
METHOD PUBLIC CyclicLogic
//! @description This method should be called cyclically by descendant function blocks by invoking <c>SUPER^.CyclicLogic()</c>.  Alternatively, the contents of this method could be reimplemented entirely in which case a call to this method would not be necessary.
VAR_Inst
	i : UDINT;
END_VAR
//Update Xplanar system status
XPlanar.Environment.Update();
XPlanar.Group.Update();

//Update Internal Mover state - Must be called every cycle 
FOR i := 1 TO SystemParameters.MOVER_COUNT DO
	IF ip.Movers[i] <> 0 THEN
		ip.Movers[i].pm.Update();
	END_IF
END_FOR

//Update INTERNAL Track status - Must be called every cycle 
FOR i := 1 TO SystemParameters.TRACK_COUNT DO
	IF ip.Tracks[i] <> 0 THEN
		ip.Tracks[i].pm.Update();
	END_IF
END_FOR

EnablePlanarGroup.Update();
MoverDetection.Update();
MoverIdentification.Update();
XPlanarReset.Update();

FOR i := 1 TO XPlanar.PartCount DO
	Parts[i].CyclicLogic();
END_FOR

//Make sure things are initialized
IF NOT _InitComplete THEN
	_InitComplete := Initialize();
	RETURN;
END_IF

//Update Mover status
FOR i := 1 TO SystemParameters.MOVER_COUNT DO
	IF ipMoverCyclic[i] <> 0 THEN
		ipMoverCyclic[i].CyclicLogic();
	END_IF
END_FOR

//Update Track status 
FOR i := 1 TO SystemParameters.TRACK_COUNT DO
	IF ipTrackCyclic[i] <> 0 THEN
		ipTrackCyclic[i].CyclicLogic();
	END_IF
END_FOR

//Update Station IDs
FOR i := 1 TO SystemParameters.STATION_COUNT DO
	IF ip.Stations[i] <> 0 THEN
		ip.Stations[i].ID := i;
	END_IF
END_FOR

FOR i := 1 TO XPlanar.TileCount DO
	Tiles[i].CyclicLogic();
END_FOR

